C07414=1103.558,-13.554,-51.728,179.876,6.251,149.168
C07415=1103.552,-13.305,-51.741,179.876,6.255,149.169
C07416=1103.547,-13.056,-51.756,179.877,6.260,149.169
C07417=1103.543,-12.806,-51.769,179.877,6.265,149.170
C07418=1103.538,-12.557,-51.784,179.878,6.269,149.171
C07419=1103.532,-12.308,-51.798,179.878,6.273,149.172
C07420=1103.527,-12.058,-51.812,179.879,6.278,149.173
C07421=1103.522,-11.808,-51.826,179.879,6.283,149.174
C07422=1103.518,-11.558,-51.840,179.880,6.287,149.175
C07423=1103.512,-11.309,-51.854,179.880,6.292,149.175
C07424=1103.507,-11.060,-51.869,179.881,6.296,149.176
C07425=1103.502,-10.810,-51.883,179.881,6.300,149.177
C07426=1103.497,-10.560,-51.897,179.881,6.305,149.178
C07427=1103.492,-10.311,-51.911,179.882,6.310,149.179
C07428=1103.487,-10.062,-51.925,179.882,6.314,149.180
C07429=1103.482,-9.812,-51.939,179.883,6.319,149.180
C07430=1103.477,-9.562,-51.953,179.884,6.323,149.181
C07431=1103.472,-9.313,-51.968,179.884,6.327,149.182
C07432=1103.467,-9.063,-51.982,179.884,6.332,149.183
C07433=1103.463,-8.813,-51.996,179.885,6.337,149.184
C07434=1103.457,-8.564,-52.010,179.886,6.341,149.185
C07435=1103.452,-8.315,-52.024,179.886,6.346,149.186
C07436=1103.447,-8.065,-52.039,179.887,6.351,149.186
C07437=1103.442,-7.815,-52.053,179.887,6.354,149.187
C07438=1103.437,-7.565,-52.067,179.888,6.359,149.188
C07439=1103.432,-7.316,-52.081,179.888,6.364,149.189
C07440=1103.427,-7.067,-52.096,179.889,6.368,149.190
C07441=1103.422,-6.818,-52.110,179.889,6.373,149.191
C07442=1103.416,-6.568,-52.125,179.890,6.377,149.191
C07443=1103.411,-6.318,-52.140,179.891,6.382,149.192
C07444=1103.406,-6.068,-52.154,179.891,6.386,149.193
C07445=1103.401,-5.819,-52.168,179.891,6.391,149.194
C07446=1103.396,-5.570,-52.182,179.892,6.395,149.195
C07447=1103.391,-5.320,-52.197,179.893,6.400,149.196
C07448=1103.386,-5.071,-52.211,179.893,6.404,149.197
C07449=1103.382,-4.857,-52.223,179.894,6.408,149.197
C07450=1103.378,-4.642,-52.236,179.895,6.412,149.198
C07451=1103.374,-4.429,-52.248,179.895,6.416,149.199
C07452=1103.369,-4.215,-52.260,179.895,6.419,149.199
C07453=1103.365,-4.000,-52.273,179.896,6.424,149.200
C07454=1103.361,-3.787,-52.286,179.896,6.428,149.201
C07455=1103.356,-3.573,-52.298,179.897,6.431,149.201
C07456=1103.352,-3.359,-52.310,179.898,6.435,149.202
C07457=1103.347,-3.109,-52.325,179.898,6.439,149.203
C07458=1103.342,-2.860,-52.340,179.898,6.444,149.204
C07459=1103.337,-2.610,-52.354,179.899,6.448,149.205
C07460=1103.331,-2.360,-52.369,179.900,6.453,149.205
C07461=1103.327,-2.111,-52.384,179.900,6.458,149.206
C07462=1103.322,-1.861,-52.398,179.901,6.463,149.207
C07463=1103.317,-1.612,-52.412,179.902,6.467,149.208
C07464=1103.312,-1.363,-52.427,179.902,6.472,149.209
C07465=1103.307,-1.113,-52.442,179.903,6.476,149.210
C07466=1103.302,-0.863,-52.456,179.904,6.481,149.210
C07467=1103.297,-0.614,-52.471,179.904,6.485,149.211
C07468=1103.292,-0.364,-52.486,179.905,6.490,149.212
C07469=1103.287,-0.114,-52.500,179.905,6.494,149.213
C07470=1103.282,0.135,-52.516,179.906,6.498,149.214
C07471=1103.276,0.384,-52.529,179.906,6.503,149.215
C07472=1103.271,0.633,-52.544,179.907,6.508,149.216
C07473=1103.266,0.883,-52.559,179.908,6.512,149.216
C07474=1103.261,1.133,-52.574,179.908,6.517,149.217
C07475=1103.256,1.382,-52.589,179.909,6.521,149.218
C07476=1103.251,1.632,-52.603,179.910,6.526,149.219
C07477=1103.247,1.881,-52.618,179.910,6.530,149.220
C07478=1103.241,2.131,-52.633,179.911,6.535,149.220
C07479=1103.236,2.380,-52.648,179.911,6.540,149.221
C07480=1103.232,2.630,-52.662,179.912,6.544,149.222
C07481=1103.227,2.879,-52.677,179.913,6.549,149.223
C07482=1103.221,3.129,-52.692,179.913,6.554,149.224
C07483=1103.217,3.378,-52.707,179.915,6.558,149.224
C07484=1103.212,3.628,-52.721,179.915,6.563,149.225
C07485=1103.206,3.878,-52.737,179.916,6.567,149.226
C07486=1103.202,4.127,-52.751,179.916,6.572,149.227
C07487=1103.197,4.376,-52.766,179.917,6.576,149.228
C07488=1103.191,4.626,-52.782,179.918,6.581,149.229
C07489=1103.187,4.875,-52.796,179.918,6.586,149.230
C07490=1103.182,5.125,-52.811,179.919,6.590,149.230
C07491=1103.176,5.375,-52.826,179.920,6.595,149.231
C07492=1103.172,5.624,-52.841,179.920,6.600,149.232
C07493=1103.166,5.873,-52.857,179.921,6.604,149.233
C07494=1103.161,6.123,-52.871,179.922,6.609,149.234
C07495=1103.157,6.372,-52.886,179.922,6.613,149.234
C07496=1103.151,6.622,-52.901,179.923,6.618,149.235
C07497=1103.147,6.872,-52.916,179.923,6.623,149.236
C07498=1103.141,7.121,-52.932,179.924,6.627,149.237
C07499=1103.136,7.371,-52.946,179.925,6.632,149.238
C07500=1103.132,7.620,-52.961,179.926,6.636,149.239
C07501=1103.126,7.869,-52.977,179.926,6.641,149.240
C07502=1103.122,8.118,-52.992,179.927,6.645,149.240
C07503=1103.116,8.368,-53.006,179.928,6.650,149.241
C07504=1103.111,8.617,-53.021,179.929,6.656,149.242
C07505=1103.107,8.832,-53.035,179.929,6.659,149.243
C07506=1103.103,9.046,-53.047,179.929,6.663,149.244
C07507=1103.099,9.260,-53.060,179.930,6.667,149.244
C07508=1103.094,9.473,-53.074,179.930,6.671,149.245
C07509=1103.090,9.687,-53.086,179.930,6.674,149.246
C07510=1103.086,9.901,-53.100,179.930,6.678,149.247
C07511=1103.081,10.115,-53.112,179.931,6.682,149.247
C07512=1103.077,10.329,-53.126,179.931,6.686,149.248
C07513=1103.072,10.578,-53.141,179.931,6.690,149.249
C07514=1103.067,10.828,-53.156,179.932,6.694,149.250
C07515=1103.062,11.077,-53.171,179.932,6.699,149.251
C07516=1103.057,11.327,-53.186,179.932,6.703,149.252
C07517=1103.053,11.577,-53.202,179.933,6.708,149.252
C07518=1103.047,11.826,-53.217,179.933,6.712,149.253
C07519=1103.043,12.075,-53.232,179.933,6.716,149.254
C07520=1103.037,12.325,-53.248,179.934,6.721,149.255
C07521=1103.033,12.574,-53.263,179.934,6.726,149.256
C07522=1103.027,12.824,-53.278,179.934,6.730,149.257
C07523=1103.022,13.074,-53.294,179.935,6.734,149.258
C07524=1103.017,13.323,-53.309,179.936,6.739,149.259
C07525=1103.012,13.572,-53.324,179.936,6.743,149.259
C07526=1103.007,13.821,-53.339,179.936,6.747,149.260
C07527=1103.003,14.071,-53.355,179.936,6.751,149.261
C07528=1102.998,14.321,-53.370,179.937,6.756,149.262
C07529=1102.993,14.570,-53.386,179.938,6.761,149.263
C07530=1102.987,14.819,-53.401,179.937,6.765,149.264
C07531=1102.983,15.069,-53.417,179.939,6.769,149.264
C07532=1102.978,15.319,-53.432,179.939,6.774,149.265
C07533=1102.972,15.568,-53.448,179.939,6.777,149.266
C07534=1102.968,15.817,-53.463,179.940,6.782,149.267
C07535=1102.962,16.066,-53.478,179.941,6.787,149.268
C07536=1102.958,16.316,-53.494,179.941,6.790,149.269
C07537=1102.953,16.566,-53.509,179.941,6.795,149.270
C07538=1102.947,16.815,-53.525,179.942,6.800,149.270
C07539=1102.943,17.065,-53.540,179.942,6.803,149.271
C07540=1102.938,17.314,-53.556,179.943,6.808,149.272
C07541=1102.933,17.564,-53.572,179.943,6.813,149.273
C07542=1102.928,17.813,-53.587,179.944,6.816,149.273
C07543=1102.923,18.063,-53.602,179.944,6.821,149.274
C07544=1102.918,18.312,-53.618,179.944,6.825,149.275
C07545=1102.912,18.562,-53.634,179.945,6.830,149.276
C07546=1102.908,18.811,-53.649,179.946,6.834,149.277
C07547=1102.903,19.061,-53.665,179.946,6.838,149.278
C07548=1102.898,19.310,-53.680,179.947,6.842,149.278
C07549=1102.893,19.559,-53.695,179.947,6.847,149.279
C07550=1102.888,19.809,-53.711,179.947,6.851,149.280
C07551=1102.883,20.058,-53.727,179.948,6.855,149.281
C07552=1102.878,20.308,-53.743,179.949,6.860,149.282
C07553=1102.874,20.557,-53.758,179.949,6.864,149.283
C07554=1102.868,20.807,-53.774,179.950,6.868,149.283
C07555=1102.863,21.056,-53.790,179.951,6.873,149.284
C07556=1102.858,21.306,-53.805,179.951,6.876,149.285
C07557=1102.853,21.555,-53.820,179.952,6.881,149.286
C07558=1102.848,21.804,-53.837,179.952,6.884,149.286
C07559=1102.844,22.054,-53.853,179.953,6.889,149.287
C07560=1102.838,22.304,-53.868,179.954,6.893,149.288
C07561=1102.835,22.518,-53.881,179.954,6.897,149.289
C07562=1102.830,22.731,-53.895,179.954,6.900,149.289
C07563=1102.826,22.945,-53.909,179.955,6.904,149.290
C07564=1102.822,23.158,-53.922,179.955,6.908,149.291
C07565=1102.817,23.373,-53.936,179.956,6.911,149.291
C07566=1102.812,23.586,-53.949,179.956,6.915,149.292
C07567=1102.808,23.800,-53.963,179.957,6.919,149.292
C07568=1102.805,24.014,-53.977,179.958,6.922,149.293
C07569=1102.800,24.263,-53.992,179.958,6.926,149.294
C07570=1102.794,24.513,-54.008,179.959,6.931,149.295
C07571=1102.790,24.762,-54.024,179.959,6.935,149.296
C07572=1102.784,25.012,-54.040,179.960,6.939,149.296
C07573=1102.779,25.262,-54.056,179.960,6.943,149.297
C07574=1102.775,25.510,-54.072,179.961,6.948,149.298
C07575=1102.770,25.760,-54.087,179.961,6.952,149.299
C07576=1102.765,26.010,-54.103,179.962,6.956,149.299
C07577=1102.760,26.258,-54.119,179.963,6.960,149.300
C07578=1102.755,26.509,-54.135,179.963,6.964,149.301
C07579=1102.750,26.758,-54.151,179.964,6.969,149.302
C07580=1102.745,27.007,-54.167,179.965,6.972,149.302
C07581=1102.740,27.257,-54.183,179.965,6.977,149.303
C07582=1102.734,27.506,-54.199,179.966,6.981,149.304
C07583=1102.730,27.756,-54.216,179.966,6.985,149.305
C07584=1102.725,28.005,-54.231,179.967,6.989,149.305
C07585=1102.721,28.254,-54.247,179.969,6.994,149.306
C07586=1102.715,28.504,-54.263,179.968,6.997,149.307
C07587=1102.711,28.753,-54.279,179.970,7.002,149.307
C07588=1102.706,29.003,-54.295,179.971,7.006,149.308
C07589=1102.700,29.252,-54.311,179.971,7.010,149.309
C07590=1102.696,29.502,-54.327,179.972,7.014,149.310
C07591=1102.690,29.751,-54.343,179.973,7.019,149.310
C07592=1102.686,30.000,-54.360,179.973,7.022,149.311
C07593=1102.680,30.250,-54.375,179.974,7.027,149.312
C07594=1102.676,30.499,-54.392,179.974,7.030,149.313
C07595=1102.671,30.749,-54.407,179.975,7.035,149.313
C07596=1102.666,30.998,-54.424,179.976,7.039,149.314
C07597=1102.661,31.248,-54.440,179.976,7.043,149.315
C07598=1102.656,31.497,-54.456,179.977,7.047,149.315
C07599=1102.651,31.746,-54.473,179.978,7.051,149.316
C07600=1102.646,31.996,-54.489,179.979,7.055,149.317
C07601=1102.641,32.245,-54.505,179.980,7.059,149.317
C07602=1102.637,32.495,-54.521,179.980,7.064,149.318
C07603=1102.631,32.744,-54.537,179.981,7.067,149.319
C07604=1102.627,32.994,-54.553,179.982,7.072,149.320
C07605=1102.621,33.243,-54.570,179.983,7.076,149.320
C07606=1102.616,33.492,-54.587,179.983,7.080,149.321
C07607=1102.612,33.742,-54.603,179.984,7.084,149.322
C07608=1102.606,33.991,-54.619,179.985,7.089,149.322
C07609=1102.602,34.241,-54.636,179.986,7.092,149.323
C07610=1102.597,34.490,-54.651,179.987,7.096,149.324
C07611=1102.592,34.740,-54.668,179.988,7.101,149.324
C07612=1102.587,34.989,-54.683,179.988,7.104,149.325
C07613=1102.582,35.238,-54.700,179.989,7.109,149.326
C07614=1102.576,35.488,-54.717,179.990,7.113,149.326
C07615=1102.572,35.737,-54.734,179.990,7.117,149.327
C07616=1102.567,35.987,-54.750,179.991,7.121,149.328
C07617=1102.563,36.200,-54.764,179.992,7.124,149.328
C07618=1102.559,36.414,-54.778,179.993,7.128,149.329
C07619=1102.554,36.628,-54.792,179.993,7.131,149.330
C07620=1102.550,36.841,-54.806,179.994,7.134,149.330
C07621=1102.546,37.055,-54.820,179.995,7.139,149.331
C07622=1102.541,37.269,-54.834,179.996,7.142,149.331
C07623=1102.537,37.483,-54.848,179.996,7.145,149.332
C07624=1102.533,37.696,-54.862,179.997,7.149,149.332
C07625=1102.528,37.946,-54.878,179.998,7.153,149.333
C07626=1102.524,38.195,-54.895,179.998,7.157,149.334
C07627=1102.519,38.444,-54.911,180.000,7.161,149.334
C07628=1102.514,38.694,-54.928,-179.999,7.165,149.335
C07629=1102.509,38.944,-54.945,-179.999,7.169,149.336
C07630=1102.503,39.193,-54.961,-179.998,7.173,149.336
C07631=1102.499,39.442,-54.978,-179.997,7.177,149.337
C07632=1102.494,39.691,-54.994,-179.996,7.181,149.338
C07633=1102.489,39.941,-55.011,-179.995,7.185,149.338
C07634=1102.484,40.190,-55.028,-179.994,7.189,149.339
C07635=1102.479,40.439,-55.044,-179.994,7.193,149.340
C07636=1102.475,40.689,-55.061,-179.993,7.197,149.340
C07637=1102.469,40.939,-55.077,-179.992,7.202,149.341
C07638=1102.464,41.188,-55.094,-179.991,7.205,149.342
C07639=1102.460,41.437,-55.110,-179.990,7.209,149.342
C07640=1102.454,41.687,-55.128,-179.989,7.213,149.343
C07641=1102.449,41.936,-55.144,-179.988,7.217,149.343
C07642=1102.445,42.185,-55.161,-179.987,7.221,149.344
C07643=1102.440,42.435,-55.177,-179.986,7.225,149.345
C07644=1102.434,42.684,-55.194,-179.985,7.229,149.345
C07645=1102.430,42.934,-55.211,-179.984,7.233,149.346
C07646=1102.425,43.183,-55.227,-179.983,7.238,149.347
C07647=1102.420,43.433,-55.245,-179.983,7.241,149.347
C07648=1102.415,43.682,-55.261,-179.982,7.245,149.348
C07649=1102.411,43.931,-55.278,-179.980,7.249,149.348
C07650=1102.405,44.181,-55.295,-179.980,7.253,149.349
C07651=1102.400,44.430,-55.311,-179.979,7.257,149.350
C07652=1102.396,44.679,-55.328,-179.978,7.261,149.350
C07653=1102.391,44.929,-55.345,-179.977,7.266,149.351
C07654=1102.386,45.178,-55.362,-179.976,7.269,149.352
C07655=1102.380,45.428,-55.379,-179.975,7.274,149.352
C07656=1102.376,45.677,-55.395,-179.973,7.277,149.353
C07657=1102.371,45.926,-55.412,-179.973,7.281,149.353
C07658=1102.366,46.176,-55.429,-179.972,7.285,149.354
C07659=1102.361,46.424,-55.446,-179.971,7.290,149.355
C07660=1102.356,46.674,-55.464,-179.970,7.293,149.355
C07661=1102.352,46.924,-55.480,-179.969,7.297,149.356
C07662=1102.347,47.173,-55.497,-179.968,7.301,149.357
C07663=1102.341,47.422,-55.514,-179.967,7.305,149.357
C07664=1102.337,47.672,-55.531,-179.966,7.309,149.358
C07665=1102.332,47.922,-55.548,-179.965,7.313,149.359
C07666=1102.328,48.170,-55.565,-179.964,7.317,149.359
C07667=1102.322,48.420,-55.582,-179.963,7.321,149.360
C07668=1102.317,48.669,-55.599,-179.962,7.325,149.360
C07669=1102.312,48.919,-55.616,-179.961,7.329,149.361
C07670=1102.308,49.168,-55.633,-179.960,7.333,149.361
C07671=1102.303,49.417,-55.651,-179.959,7.337,149.362
C07672=1102.298,49.667,-55.667,-179.958,7.341,149.363
C07673=1102.294,49.878,-55.681,-179.957,7.344,149.363
C07674=1102.290,50.089,-55.696,-179.956,7.348,149.364
C07675=1102.285,50.301,-55.710,-179.955,7.351,149.364
C07676=1102.281,50.512,-55.726,-179.955,7.354,149.365
C07677=1102.277,50.724,-55.739,-179.953,7.358,149.365
C07678=1102.273,50.934,-55.754,-179.953,7.361,149.366
C07679=1102.269,51.146,-55.768,-179.952,7.365,149.366
C07680=1102.265,51.357,-55.783,-179.951,7.368,149.367
C07681=1102.259,51.607,-55.800,-179.950,7.372,149.367
C07682=1102.255,51.855,-55.818,-179.949,7.375,149.368
C07683=1102.250,52.105,-55.835,-179.948,7.379,149.368
C07684=1102.245,52.355,-55.852,-179.946,7.384,149.369
C07685=1102.240,52.605,-55.869,-179.945,7.388,149.370
C07686=1102.235,52.854,-55.887,-179.944,7.391,149.370
C07687=1102.231,53.103,-55.903,-179.943,7.395,149.371
C07688=1102.226,53.352,-55.921,-179.942,7.400,149.371
C07689=1101.999,43.459,-55.292,-179.978,7.245,149.347
C07690=1102.004,43.210,-55.276,-179.979,7.240,149.346
C07691=1102.009,42.960,-55.259,-179.980,7.236,149.345
C07692=1102.013,42.710,-55.242,-179.981,7.232,149.345
C07693=1102.018,42.461,-55.225,-179.981,7.228,149.344
C07694=1102.024,42.212,-55.208,-179.983,7.224,149.343
C07695=1102.028,41.962,-55.192,-179.984,7.220,149.343
C07696=1102.033,41.713,-55.175,-179.984,7.216,149.342
C07697=1102.038,41.464,-55.158,-179.985,7.212,149.341
C07698=1102.043,41.214,-55.141,-179.987,7.208,149.341
C07699=1102.047,40.965,-55.125,-179.987,7.204,149.340
C07700=1102.052,40.716,-55.108,-179.988,7.200,149.340
C07701=1102.058,40.466,-55.091,-179.989,7.196,149.339
C07702=1102.062,40.217,-55.074,-179.990,7.192,149.338
C07703=1102.068,39.967,-55.059,-179.991,7.188,149.338
C07704=1102.072,39.718,-55.042,-179.992,7.184,149.337
C07705=1102.077,39.468,-55.025,-179.992,7.180,149.336
C07706=1102.082,39.219,-55.009,-179.993,7.176,149.336
C07707=1102.087,38.970,-54.992,-179.994,7.172,149.335
C07708=1102.091,38.720,-54.975,-179.995,7.168,149.334
C07709=1102.097,38.471,-54.959,-179.996,7.164,149.334
C07710=1102.102,38.221,-54.942,-179.996,7.160,149.333
C07711=1102.107,37.972,-54.926,-179.998,7.156,149.332
C07712=1102.111,37.723,-54.909,-179.999,7.152,149.332
C07713=1102.116,37.473,-54.893,-179.999,7.148,149.331
C07714=1102.123,37.103,-54.868,180.000,7.141,149.330
C07715=1102.131,36.733,-54.844,179.999,7.136,149.329
C07716=1102.138,36.363,-54.819,179.997,7.129,149.328
C07717=1102.146,35.993,-54.795,179.996,7.123,149.327
C07718=1102.151,35.743,-54.779,179.995,7.119,149.326
C07719=1102.156,35.494,-54.762,179.995,7.116,149.326
C07720=1102.161,35.245,-54.746,179.994,7.111,149.325
C07721=1102.165,34.996,-54.729,179.993,7.107,149.324
C07722=1102.171,34.746,-54.714,179.992,7.104,149.324
C07723=1102.175,34.497,-54.697,179.991,7.099,149.323
C07724=1102.181,34.248,-54.680,179.991,7.095,149.322
C07725=1102.186,33.998,-54.664,179.990,7.091,149.322
C07726=1102.190,33.748,-54.648,179.989,7.087,149.321
C07727=1102.196,33.499,-54.632,179.988,7.082,149.320
C07728=1102.200,33.249,-54.615,179.987,7.079,149.320
C07729=1102.205,33.000,-54.599,179.986,7.075,149.319
C07730=1102.210,32.750,-54.583,179.986,7.070,149.318
C07731=1102.215,32.501,-54.567,179.985,7.066,149.317
C07732=1102.219,32.252,-54.550,179.984,7.062,149.317
C07733=1102.225,32.003,-54.534,179.983,7.058,149.316
C07734=1102.229,31.753,-54.518,179.983,7.054,149.315
C07735=1102.235,31.504,-54.502,179.982,7.050,149.314
C07736=1102.239,31.254,-54.486,179.982,7.046,149.314
C07737=1102.245,31.005,-54.470,179.981,7.042,149.313
C07738=1102.250,30.755,-54.453,179.980,7.037,149.313
C07739=1102.255,30.506,-54.437,179.980,7.034,149.312
C07740=1102.260,30.256,-54.420,179.979,7.029,149.311
C07741=1102.265,30.007,-54.405,179.978,7.025,149.310
C07742=1102.270,29.757,-54.388,179.977,7.021,149.310
C07743=1102.275,29.508,-54.373,179.977,7.017,149.309
C07744=1102.279,29.258,-54.356,179.975,7.012,149.308
C07745=1102.284,29.009,-54.341,179.975,7.009,149.307
C07746=1102.289,28.760,-54.324,179.974,7.004,149.307
C07747=1102.294,28.510,-54.309,179.973,7.000,149.306
C07748=1102.298,28.261,-54.292,179.973,6.996,149.305
C07749=1102.304,28.011,-54.276,179.972,6.992,149.304
C07750=1102.308,27.762,-54.260,179.972,6.988,149.304
C07751=1102.314,27.513,-54.244,179.971,6.984,149.303
C07752=1102.319,27.263,-54.229,179.970,6.979,149.302
C07753=1102.324,27.014,-54.212,179.970,6.976,149.302
C07754=1102.329,26.764,-54.196,179.969,6.971,149.301
C07755=1102.333,26.515,-54.180,179.968,6.967,149.300
C07756=1102.339,26.265,-54.164,179.968,6.963,149.299
C07757=1102.344,26.015,-54.148,179.967,6.958,149.298
C07758=1102.349,25.767,-54.132,179.966,6.954,149.298
C07759=1102.354,25.517,-54.116,179.966,6.951,149.297
C07760=1102.358,25.267,-54.101,179.965,6.946,149.296
C07761=1102.363,25.019,-54.085,179.965,6.942,149.296
C07762=1102.368,24.768,-54.069,179.964,6.938,149.295
C07763=1102.373,24.519,-54.053,179.963,6.933,149.294
C07764=1102.378,24.270,-54.037,179.963,6.929,149.293
C07765=1102.383,24.020,-54.021,179.962,6.925,149.292
C07766=1102.387,23.807,-54.008,179.962,6.922,149.292
C07767=1102.391,23.593,-53.994,179.961,6.918,149.291
C07768=1102.396,23.379,-53.980,179.961,6.915,149.290
C07769=1102.401,23.165,-53.967,179.960,6.911,149.290
C07770=1102.404,22.951,-53.953,179.959,6.907,149.289
C07771=1102.409,22.738,-53.939,179.959,6.903,149.289
C07772=1102.413,22.524,-53.926,179.958,6.900,149.288
C07773=1102.417,22.311,-53.913,179.958,6.896,149.287
C07774=1102.422,22.060,-53.897,179.957,6.892,149.286
C07775=1102.427,21.811,-53.881,179.957,6.888,149.286
C07776=1102.432,21.562,-53.865,179.956,6.883,149.285
C07777=1102.436,21.313,-53.850,179.956,6.880,149.284
C07778=1102.442,21.063,-53.834,179.955,6.875,149.283
C07779=1102.447,20.813,-53.818,179.955,6.870,149.282
C07780=1102.452,20.564,-53.803,179.954,6.867,149.282
C07781=1102.457,20.315,-53.786,179.954,6.862,149.281
C07782=1102.461,20.065,-53.771,179.953,6.858,149.280
C07783=1102.466,19.816,-53.755,179.953,6.854,149.279
C07784=1102.472,19.566,-53.740,179.952,6.849,149.278
C07785=1102.477,19.317,-53.724,179.952,6.846,149.278
C07786=1102.481,19.067,-53.709,179.951,6.841,149.277
C07787=1102.487,18.818,-53.693,179.951,6.836,149.276
C07788=1102.492,18.568,-53.678,179.950,6.833,149.275
C07789=1102.496,18.319,-53.662,179.950,6.828,149.274
C07790=1102.501,18.070,-53.646,179.949,6.823,149.273
C07791=1102.507,17.820,-53.630,179.949,6.820,149.273
C07792=1102.511,17.570,-53.614,179.948,6.815,149.272
C07793=1102.516,17.321,-53.599,179.948,6.810,149.271
C07794=1102.521,17.072,-53.584,179.947,6.807,149.270
C07795=1102.527,16.822,-53.568,179.947,6.802,149.270
C07796=1102.531,16.572,-53.553,179.947,6.798,149.269
C07797=1102.536,16.323,-53.537,179.946,6.794,149.268
C07798=1102.542,16.074,-53.522,179.945,6.789,149.267
C07799=1102.546,15.825,-53.507,179.945,6.785,149.266
C07800=1102.551,15.574,-53.491,179.945,6.781,149.265
C07801=1102.556,15.325,-53.475,179.944,6.776,149.264
C07802=1102.561,15.076,-53.460,179.944,6.772,149.264
C07803=1102.566,14.827,-53.445,179.943,6.768,149.263
C07804=1102.571,14.577,-53.429,179.942,6.763,149.262
C07805=1102.576,14.327,-53.414,179.943,6.759,149.261
C07806=1102.581,14.078,-53.398,179.942,6.754,149.260
C07807=1102.586,13.829,-53.383,179.941,6.750,149.259
C07808=1102.591,13.579,-53.367,179.941,6.746,149.259
C07809=1102.595,13.330,-53.352,179.940,6.742,149.258
C07810=1102.601,13.080,-53.337,179.940,6.738,149.257
C07811=1102.606,12.830,-53.322,179.940,6.733,149.256
C07812=1102.611,12.581,-53.307,179.939,6.728,149.255
C07813=1102.616,12.331,-53.291,179.939,6.724,149.254
C07814=1102.621,12.082,-53.276,179.939,6.720,149.253
C07815=1102.626,11.833,-53.260,179.938,6.715,149.252
C07816=1102.631,11.583,-53.245,179.938,6.711,149.252
C07817=1102.636,11.334,-53.230,179.938,6.706,149.251
C07818=1102.640,11.084,-53.215,179.937,6.702,149.250
C07819=1102.646,10.834,-53.199,179.937,6.698,149.249
C07820=1102.651,10.585,-53.184,179.936,6.693,149.248
C07821=1102.656,10.336,-53.169,179.936,6.689,149.247
C07822=1102.659,10.122,-53.156,179.936,6.685,149.246
C07823=1102.664,9.908,-53.142,179.935,6.681,149.246
C07824=1102.669,9.694,-53.130,179.935,6.677,149.245
C07825=1102.673,9.480,-53.117,179.935,6.674,149.244
C07826=1102.677,9.267,-53.104,179.935,6.670,149.243
C07827=1102.681,9.052,-53.090,179.935,6.666,149.243
C07828=1102.686,8.839,-53.077,179.935,6.662,149.242
C07829=1102.690,8.625,-53.065,179.934,6.658,149.241
C07830=1102.695,8.375,-53.049,179.933,6.653,149.240
C07831=1102.699,8.126,-53.034,179.933,6.649,149.239
C07832=1102.705,7.876,-53.019,179.932,6.644,149.239
C07833=1102.710,7.627,-53.005,179.931,6.640,149.238
C07834=1102.715,7.377,-52.989,179.931,6.635,149.237
C07835=1102.720,7.128,-52.974,179.930,6.630,149.236
C07836=1102.726,6.878,-52.959,179.929,6.626,149.235
C07837=1102.730,6.629,-52.944,179.928,6.621,149.234
C07838=1102.734,6.379,-52.929,179.928,6.617,149.234
C07839=1102.740,6.129,-52.914,179.927,6.612,149.233
C07840=1102.745,5.880,-52.899,179.926,6.608,149.232
C07841=1102.750,5.631,-52.883,179.926,6.603,149.231
C07842=1102.755,5.381,-52.869,179.925,6.598,149.230
C07843=1102.760,5.132,-52.854,179.924,6.594,149.230
C07844=1102.765,4.883,-52.838,179.924,6.589,149.229
C07845=1102.770,4.633,-52.824,179.923,6.584,149.228
C07846=1102.775,4.384,-52.809,179.923,6.580,149.227
C07847=1102.780,4.134,-52.794,179.922,6.575,149.226
C07848=1102.785,3.885,-52.779,179.921,6.571,149.225
C07849=1102.791,3.635,-52.764,179.921,6.566,149.224
C07850=1102.795,3.386,-52.749,179.920,6.561,149.224
C07851=1102.800,3.137,-52.734,179.919,6.557,149.223
C07852=1102.805,2.886,-52.719,179.919,6.552,149.222
C07853=1102.810,2.637,-52.704,179.918,6.547,149.221
C07854=1102.815,2.387,-52.690,179.917,6.543,149.220
C07855=1102.819,2.138,-52.675,179.916,6.538,149.220
C07856=1102.825,1.888,-52.660,179.916,6.534,149.219
C07857=1102.830,1.639,-52.645,179.915,6.529,149.218
C07858=1102.835,1.389,-52.631,179.914,6.525,149.217
C07859=1102.840,1.139,-52.616,179.914,6.520,149.216
C07860=1102.845,0.890,-52.601,179.913,6.515,149.215
C07861=1102.850,0.640,-52.587,179.912,6.511,149.215
C07862=1102.854,0.391,-52.572,179.912,6.506,149.214
C07863=1102.860,0.141,-52.557,179.911,6.502,149.213
C07864=1102.865,-0.108,-52.542,179.910,6.497,149.212
C07865=1102.870,-0.358,-52.527,179.910,6.492,149.211
C07866=1102.875,-0.607,-52.513,179.909,6.488,149.210
C07867=1102.880,-0.857,-52.498,179.909,6.483,149.209
C07868=1102.885,-1.107,-52.483,179.908,6.480,149.209
C07869=1102.890,-1.355,-52.469,179.908,6.475,149.208
C07870=1102.895,-1.605,-52.454,179.907,6.470,149.207
C07871=1102.900,-1.854,-52.440,179.906,6.466,149.206
C07872=1102.906,-2.104,-52.425,179.906,6.461,149.205
C07873=1102.911,-2.353,-52.410,179.905,6.456,149.205
C07874=1102.916,-2.603,-52.396,179.904,6.452,149.204
C07875=1102.920,-2.852,-52.381,179.904,6.447,149.203
C07876=1102.925,-3.102,-52.367,179.903,6.443,149.202
C07877=1102.930,-3.352,-52.352,179.903,6.438,149.201
C07878=1102.935,-3.565,-52.339,179.902,6.434,149.201
C07879=1102.939,-3.780,-52.327,179.902,6.431,149.200
C07880=1102.943,-3.994,-52.315,179.901,6.426,149.199
C07881=1102.948,-4.208,-52.303,179.900,6.423,149.199
C07882=1102.952,-4.421,-52.290,179.901,6.419,149.198
C07883=1102.956,-4.636,-52.278,179.900,6.415,149.197
C07884=1102.960,-4.850,-52.266,179.899,6.411,149.196
C07885=1102.964,-5.063,-52.253,179.899,6.408,149.196
C07886=1102.970,-5.313,-52.238,179.898,6.403,149.195
C07887=1102.975,-5.563,-52.224,179.898,6.398,149.194
C07888=1102.980,-5.812,-52.209,179.897,6.394,149.193
C07889=1102.985,-6.061,-52.194,179.896,6.389,149.192
C07890=1102.990,-6.310,-52.180,179.896,6.384,149.191
C07891=1102.995,-6.560,-52.166,179.895,6.380,149.190
C07892=1103.000,-6.810,-52.152,179.895,6.376,149.190
C07893=1103.005,-7.060,-52.138,179.894,6.371,149.189
C07894=1103.010,-7.309,-52.123,179.894,6.367,149.188
C07895=1103.015,-7.559,-52.109,179.893,6.362,149.187
C07896=1103.020,-7.808,-52.094,179.892,6.358,149.186
C07897=1103.025,-8.057,-52.080,179.892,6.353,149.186
C07898=1103.030,-8.307,-52.066,179.891,6.348,149.185
C07899=1103.035,-8.557,-52.052,179.891,6.344,149.184
C07900=1103.040,-8.806,-52.037,179.890,6.340,149.183
C07901=1103.045,-9.056,-52.023,179.890,6.335,149.182
C07902=1103.050,-9.306,-52.009,179.889,6.331,149.181
C07903=1103.056,-9.555,-51.995,179.889,6.326,149.180
C07904=1103.060,-9.804,-51.981,179.888,6.322,149.180
C07905=1103.065,-10.054,-51.966,179.888,6.318,149.179
C07906=1103.070,-10.304,-51.952,179.887,6.313,149.178
C07907=1103.075,-10.554,-51.938,179.887,6.308,149.177
C07908=1103.081,-10.803,-51.924,179.886,6.303,149.176
C07909=1103.086,-11.052,-51.910,179.886,6.299,149.175
C07910=1103.091,-11.302,-51.895,179.885,6.294,149.175
C07911=1103.096,-11.552,-51.881,179.885,6.291,149.174
C07912=1103.101,-11.801,-51.867,179.885,6.286,149.173
C07913=1103.106,-12.050,-51.853,179.884,6.281,149.172
C07914=1103.111,-12.300,-51.839,179.884,6.276,149.171
C07915=1103.116,-12.550,-51.824,179.883,6.272,149.170
C07916=1103.120,-12.799,-51.811,179.883,6.268,149.169
C07917=1103.126,-13.048,-51.797,179.882,6.263,149.168
C07918=1103.131,-13.298,-51.782,179.882,6.259,149.168
C07919=1103.136,-13.548,-51.768,179.881,6.254,149.167
C07920=1103.141,-13.797,-51.754,179.881,6.249,149.166
C07921=1103.146,-14.046,-51.740,179.881,6.245,149.165
C07922=1103.151,-14.296,-51.726,179.880,6.241,149.164
C07923=1103.157,-14.546,-51.712,179.879,6.236,149.163
C07924=1103.161,-14.796,-51.698,179.879,6.232,149.162
C07925=1103.166,-15.045,-51.684,179.878,6.227,149.162
C07926=1103.171,-15.295,-51.670,179.878,6.223,149.161
C07927=1103.176,-15.544,-51.656,179.878,6.218,149.160
C07928=1103.181,-15.794,-51.642,179.877,6.213,149.159
C07929=1103.187,-16.043,-51.628,179.877,6.209,149.158
C07930=1103.191,-16.293,-51.615,179.876,6.204,149.157
C07931=1103.196,-16.543,-51.600,179.877,6.200,149.156
C07932=1103.202,-16.792,-51.587,179.876,6.195,149.155
C07933=1103.207,-17.041,-51.572,179.876,6.191,149.154
C07934=1103.211,-17.255,-51.560,179.875,6.187,149.154
C07935=1103.216,-17.469,-51.548,179.875,6.182,149.153
C07936=1103.220,-17.683,-51.538,179.874,6.179,149.152
C07937=1103.224,-17.897,-51.525,179.874,6.175,149.151
C07938=1103.228,-18.112,-51.513,179.874,6.171,149.150
C07939=1103.233,-18.326,-51.501,179.873,6.167,149.150
C07940=1103.237,-18.540,-51.489,179.873,6.163,149.149
C07941=1103.241,-18.754,-51.477,179.873,6.160,149.148
C07942=1103.247,-19.003,-51.464,179.872,6.155,149.147
C07943=1103.252,-19.253,-51.450,179.872,6.150,149.146
C07944=1103.256,-19.503,-51.436,179.872,6.146,149.146
C07945=1103.262,-19.752,-51.423,179.872,6.141,149.145
C07946=1103.267,-20.002,-51.409,179.871,6.137,149.144
C07947=1103.272,-20.251,-51.395,179.871,6.132,149.143
C07948=1103.277,-20.501,-51.381,179.870,6.127,149.142
C07949=1103.282,-20.751,-51.367,179.870,6.123,149.141
C07950=1103.287,-21.000,-51.354,179.870,6.118,149.140
C07951=1103.292,-21.250,-51.340,179.870,6.114,149.139
C07952=1103.297,-21.499,-51.326,179.869,6.109,149.138
C07953=1103.302,-21.748,-51.313,179.869,6.104,149.137
C07954=1103.307,-21.998,-51.299,179.869,6.100,149.136
C07955=1103.312,-22.248,-51.285,179.868,6.095,149.135
C07956=1103.318,-22.497,-51.272,179.868,6.091,149.134
C07957=1103.322,-22.747,-51.258,179.867,6.086,149.134
C07958=1103.328,-22.996,-51.244,179.867,6.081,149.132
C07959=1103.333,-23.246,-51.231,179.868,6.077,149.132
C07960=1103.338,-23.495,-51.217,179.867,6.072,149.131
C07961=1103.343,-23.746,-51.204,179.867,6.067,149.130
C07962=1103.348,-23.995,-51.190,179.866,6.063,149.129
C07963=1103.353,-24.245,-51.177,179.866,6.058,149.128
C07964=1103.358,-24.494,-51.163,179.866,6.054,149.127
C07965=1103.364,-24.744,-51.150,179.866,6.049,149.126
C07966=1103.368,-24.993,-51.136,179.865,6.044,149.125
C07967=1103.374,-25.243,-51.123,179.865,6.039,149.124
C07968=1103.379,-25.492,-51.109,179.865,6.034,149.123
C07969=1103.384,-25.742,-51.096,179.865,6.031,149.122
C07970=1103.389,-25.991,-51.082,179.865,6.026,149.121
C07971=1103.394,-26.242,-51.068,179.865,6.021,149.120
C07972=1103.399,-26.490,-51.055,179.864,6.016,149.119
C07973=1103.404,-26.741,-51.041,179.864,6.011,149.118
C07974=1103.409,-26.989,-51.028,179.864,6.007,149.117
C07975=1103.414,-27.240,-51.015,179.863,6.003,149.116
C07976=1103.419,-27.488,-51.001,179.863,5.998,149.115
C07977=1103.424,-27.739,-50.988,179.862,5.993,149.115
C07978=1103.430,-27.988,-50.975,179.862,5.988,149.114
C07979=1103.434,-28.238,-50.961,179.862,5.984,149.113
C07980=1103.440,-28.487,-50.948,179.862,5.980,149.112
C07981=1103.444,-28.737,-50.934,179.861,5.975,149.111
C07982=1103.450,-28.986,-50.921,179.861,5.970,149.110
C07983=1103.455,-29.236,-50.908,179.861,5.966,149.109
C07984=1103.460,-29.485,-50.894,179.860,5.962,149.108
C07985=1103.465,-29.735,-50.881,179.860,5.957,149.107
C07986=1103.470,-29.985,-50.868,179.859,5.952,149.106
C07987=1103.475,-30.235,-50.854,179.860,5.948,149.105
C07988=1103.480,-30.484,-50.841,179.859,5.943,149.105
C07989=1103.485,-30.734,-50.828,179.859,5.939,149.104
C07990=1103.489,-30.948,-50.816,179.858,5.935,149.103
C07991=1103.494,-31.162,-50.805,179.858,5.931,149.102
C07992=1103.498,-31.376,-50.793,179.858,5.928,149.101
C07993=1103.503,-31.590,-50.783,179.858,5.924,149.100
C07994=1103.508,-31.804,-50.771,179.857,5.919,149.100
C07995=1103.511,-32.018,-50.760,179.857,5.916,149.099
C07996=1103.516,-32.232,-50.749,179.857,5.912,149.098
C07997=1103.521,-32.446,-50.737,179.857,5.908,149.097
C07998=1103.525,-32.696,-50.724,179.856,5.904,149.097
C07999=1103.530,-32.946,-50.711,179.856,5.900,149.096
C08000=1103.536,-33.195,-50.698,179.856,5.895,149.095
C08001=1103.540,-33.445,-50.684,179.855,5.891,149.094
C08002=1103.546,-33.694,-50.671,179.855,5.887,149.093
C08003=1103.551,-33.944,-50.658,179.855,5.882,149.092
C08004=1103.556,-34.194,-50.645,179.854,5.877,149.091
C08005=1103.561,-34.444,-50.632,179.854,5.873,149.090
C08006=1103.566,-34.693,-50.619,179.854,5.869,149.090
C08007=1103.571,-34.942,-50.606,179.853,5.864,149.089
C08008=1103.576,-35.192,-50.592,179.853,5.859,149.088
C08009=1103.581,-35.442,-50.580,179.853,5.855,149.087
C08010=1103.587,-35.692,-50.566,179.853,5.851,149.086
C08011=1103.592,-35.941,-50.554,179.852,5.846,149.085
C08012=1103.597,-36.191,-50.541,179.852,5.842,149.084
C08013=1103.602,-36.440,-50.527,179.852,5.837,149.083
C08014=1103.607,-36.690,-50.514,179.852,5.832,149.082
C08015=1103.612,-36.939,-50.502,179.852,5.828,149.081
C08016=1103.617,-37.189,-50.489,179.851,5.824,149.080
C08017=1103.622,-37.439,-50.475,179.851,5.819,149.079
C08018=1103.628,-37.688,-50.463,179.851,5.815,149.079
C08019=1103.632,-37.938,-50.450,179.850,5.810,149.078
C08020=1103.638,-38.188,-50.437,179.850,5.806,149.077
C08021=1103.643,-38.437,-50.424,179.850,5.801,149.076
C08022=1103.648,-38.687,-50.411,179.850,5.797,149.075
C08023=1103.653,-38.937,-50.398,179.849,5.792,149.074
C08024=1103.659,-39.186,-50.385,179.849,5.787,149.073
C08025=1103.663,-39.436,-50.372,179.849,5.782,149.072
C08026=1103.668,-39.685,-50.360,179.849,5.778,149.071
C08027=1103.674,-39.935,-50.346,179.849,5.774,149.070
C08028=1103.679,-40.185,-50.334,179.848,5.769,149.069
C08029=1103.684,-40.434,-50.321,179.848,5.764,149.068
C08030=1103.689,-40.684,-50.308,179.848,5.759,149.067
C08031=1103.693,-40.934,-50.295,179.848,5.755,149.066
C08032=1103.699,-41.183,-50.282,179.848,5.750,149.065
C08033=1103.704,-41.433,-50.270,179.848,5.745,149.064
C08034=1103.709,-41.682,-50.257,179.847,5.741,149.063
C08035=1103.714,-41.932,-50.244,179.847,5.735,149.062
C08036=1103.720,-42.182,-50.231,179.847,5.731,149.061
C08037=1103.725,-42.431,-50.218,179.847,5.726,149.060
C08038=1103.730,-42.681,-50.205,179.847,5.722,149.059
C08039=1103.735,-42.930,-50.193,179.847,5.716,149.058
C08040=1103.740,-43.180,-50.181,179.847,5.711,149.057
C08041=1103.745,-43.429,-50.168,179.848,5.707,149.056
C08042=1103.750,-43.680,-50.155,179.847,5.702,149.055
C08043=1103.756,-43.929,-50.142,179.848,5.698,149.054
C08044=1103.761,-44.178,-50.129,179.848,5.693,149.052
C08045=1103.766,-44.428,-50.117,179.848,5.688,149.051
C08046=1103.770,-44.642,-50.106,179.848,5.684,149.050
C08047=1103.775,-44.856,-50.095,179.848,5.680,149.049
C08048=1103.779,-45.071,-50.084,179.849,5.676,149.049
C08049=1103.783,-45.285,-50.073,179.849,5.672,149.048
C08050=1103.788,-45.499,-50.062,179.849,5.668,149.047
C08051=1103.792,-45.713,-50.052,179.849,5.664,149.046
C08052=1103.796,-45.927,-50.041,179.849,5.659,149.045
C08053=1103.801,-46.142,-50.030,179.849,5.655,149.044
C08054=1103.806,-46.392,-50.018,179.850,5.651,149.043
C08055=1103.811,-46.641,-50.005,179.850,5.646,149.042
C08056=1103.817,-46.890,-49.993,179.849,5.641,149.041
C08057=1103.821,-47.140,-49.980,179.850,5.637,149.040
C08058=1103.826,-47.390,-49.967,179.850,5.632,149.038
C08059=1103.832,-47.640,-49.955,179.850,5.628,149.038
C08060=1103.837,-47.889,-49.942,179.850,5.623,149.036
C08061=1103.842,-48.138,-49.930,179.850,5.618,149.035
C08062=1103.846,-48.388,-49.917,179.851,5.613,149.034
C08063=1103.852,-48.638,-49.905,179.850,5.609,149.033
C08064=1103.857,-48.888,-49.892,179.851,5.603,149.032
C08065=1103.862,-49.137,-49.880,179.851,5.599,149.031
C08066=1103.868,-49.387,-49.868,179.851,5.594,149.030
C08067=1103.873,-49.636,-49.855,179.851,5.589,149.029
C08068=1103.877,-49.886,-49.842,179.852,5.585,149.028
C08069=1103.883,-50.136,-49.830,179.851,5.580,149.027
C08070=1103.888,-50.385,-49.818,179.851,5.575,149.026
C08071=1103.893,-50.635,-49.805,179.852,5.571,149.024
C08072=1103.898,-50.885,-49.793,179.851,5.566,149.023
C08073=1103.903,-51.134,-49.781,179.852,5.561,149.022
C08074=1103.908,-51.384,-49.768,179.852,5.557,149.021
C08075=1103.913,-51.634,-49.756,179.852,5.552,149.020
C08076=1103.918,-51.883,-49.743,179.852,5.548,149.019
C08077=1103.924,-52.133,-49.731,179.853,5.542,149.018
C08078=1103.929,-52.383,-49.719,179.852,5.538,149.017
C08079=1103.934,-52.632,-49.706,179.853,5.533,149.016
C08080=1103.940,-52.882,-49.694,179.853,5.528,149.015
C08081=1103.945,-53.131,-49.682,179.852,5.523,149.014
C08082=1103.950,-53.382,-49.669,179.853,5.519,149.013
C08083=1103.955,-53.631,-49.657,179.853,5.514,149.011
C08084=1103.960,-53.880,-49.644,179.853,5.509,149.011
C08085=1103.965,-54.130,-49.632,179.854,5.505,149.009
C08086=1103.970,-54.380,-49.620,179.854,5.500,149.008
C08087=1103.976,-54.630,-49.608,179.853,5.495,149.007
C08088=1103.981,-54.879,-49.595,179.854,5.491,149.006
C08089=1103.986,-55.129,-49.583,179.853,5.486,149.005
C08090=1103.991,-55.378,-49.571,179.854,5.481,149.004
C08091=1103.996,-55.628,-49.560,179.854,5.477,149.003
C08092=1104.001,-55.878,-49.547,179.854,5.472,149.002
C08093=1104.006,-56.128,-49.535,179.854,5.467,149.001
C08094=1104.011,-56.377,-49.522,179.855,5.462,149.000
C08095=1104.017,-56.627,-49.510,179.854,5.458,148.999
C08096=1104.022,-56.876,-49.498,179.854,5.453,148.998
C08097=1104.027,-57.126,-49.486,179.855,5.449,148.997
C08098=1104.032,-57.375,-49.474,179.855,5.443,148.996
C08099=1104.037,-57.625,-49.462,179.855,5.438,148.994
C08100=1104.042,-57.874,-49.449,179.855,5.434,148.993
C08101=1104.048,-58.124,-49.437,179.855,5.429,148.992
C08102=1104.052,-58.339,-49.427,179.855,5.425,148.991
C08103=1104.056,-58.554,-49.417,179.855,5.421,148.990
C08104=1104.061,-58.767,-49.406,179.855,5.417,148.990
C08105=1104.065,-58.982,-49.396,179.855,5.413,148.989
C08106=1104.069,-59.196,-49.386,179.855,5.409,148.988
C08107=1104.074,-59.410,-49.375,179.855,5.405,148.987
C08108=1104.078,-59.625,-49.365,179.855,5.401,148.986
C08109=1104.082,-59.839,-49.354,179.856,5.397,148.985
C08110=1104.087,-60.089,-49.343,179.855,5.393,148.984
C08111=1104.093,-60.339,-49.331,179.855,5.387,148.983
C08112=1104.098,-60.588,-49.318,179.855,5.383,148.982
C08113=1104.103,-60.838,-49.306,179.855,5.378,148.981
C08114=1104.108,-61.088,-49.295,179.855,5.373,148.980
C08115=1104.113,-61.337,-49.282,179.854,5.368,148.979
C08116=1104.119,-61.587,-49.270,179.854,5.363,148.978
C08117=1104.124,-61.837,-49.259,179.854,5.358,148.977
C08118=1104.128,-62.086,-49.247,179.854,5.353,148.976
C08119=1104.134,-62.336,-49.235,179.854,5.348,148.975
C08120=1104.139,-62.586,-49.223,179.854,5.343,148.974
C08121=1104.144,-62.834,-49.211,179.853,5.338,148.973
C08122=1104.150,-63.084,-49.199,179.853,5.333,148.972
C08123=1104.155,-63.334,-49.187,179.853,5.329,148.971
C08124=1104.161,-63.584,-49.175,179.853,5.323,148.970
C08125=1104.165,-63.833,-49.163,179.853,5.318,148.968
C08126=1104.170,-64.083,-49.152,179.853,5.314,148.967
C08127=1104.176,-64.333,-49.140,179.853,5.308,148.966
C08128=1104.180,-64.582,-49.128,179.853,5.304,148.965
C08129=1104.186,-64.832,-49.117,179.853,5.299,148.964
C08130=1104.191,-65.081,-49.104,179.853,5.293,148.963
C08131=1104.196,-65.331,-49.093,179.852,5.289,148.962
C08132=1104.201,-65.581,-49.081,179.853,5.284,148.961
C08133=1104.207,-65.831,-49.069,179.853,5.278,148.960
C08134=1104.211,-66.081,-49.058,179.852,5.274,148.959
C08135=1104.217,-66.331,-49.046,179.852,5.268,148.958
C08136=1104.222,-66.580,-49.033,179.853,5.263,148.956
C08137=1104.227,-66.829,-49.022,179.852,5.259,148.956
C08138=1104.233,-67.079,-49.010,179.852,5.253,148.954
C08139=1104.237,-67.328,-48.999,179.852,5.248,148.953
C08140=1104.243,-67.578,-48.987,179.853,5.243,148.952
C08141=1104.248,-67.828,-48.975,179.852,5.238,148.951
C08142=1104.253,-68.078,-48.964,179.852,5.233,148.950
C08143=1104.258,-68.328,-48.952,179.852,5.228,148.949
C08144=1104.263,-68.577,-48.941,179.853,5.223,148.948
C08145=1104.268,-68.827,-48.929,179.852,5.218,148.947
C08146=1104.274,-69.076,-48.918,179.852,5.213,148.946
C08147=1104.279,-69.326,-48.906,179.852,5.208,148.944
C08148=1104.284,-69.576,-48.894,179.853,5.203,148.943
C08149=1104.289,-69.826,-48.883,179.853,5.198,148.942
C08150=1104.295,-70.076,-48.871,179.853,5.193,148.941
C08151=1104.299,-70.325,-48.859,179.853,5.188,148.940
C08152=1104.305,-70.575,-48.848,179.853,5.183,148.939
C08153=1104.310,-70.824,-48.837,179.853,5.178,148.938
C08154=1104.315,-71.074,-48.825,179.853,5.172,148.936
C08155=1104.320,-71.324,-48.814,179.853,5.167,148.935
C08156=1104.326,-71.574,-48.802,179.853,5.162,148.934
C08157=1104.330,-71.823,-48.791,179.853,5.157,148.933
C08158=1104.335,-72.037,-48.780,179.853,5.152,148.932
C08159=1104.339,-72.252,-48.770,179.853,5.148,148.931
C08160=1104.344,-72.466,-48.761,179.853,5.144,148.930
C08161=1104.349,-72.681,-48.751,179.854,5.139,148.929
C08162=1104.353,-72.895,-48.741,179.853,5.135,148.928
C08163=1104.357,-73.109,-48.731,179.853,5.131,148.927
C08164=1104.362,-73.324,-48.722,179.853,5.126,148.926
C08165=1104.366,-73.538,-48.711,179.854,5.122,148.925
C08166=1104.372,-73.787,-48.701,179.853,5.117,148.924
C08167=1104.377,-74.037,-48.689,179.854,5.112,148.923
C08168=1104.382,-74.287,-48.678,179.854,5.106,148.922
C08169=1104.387,-74.537,-48.666,179.854,5.101,148.920
C08170=1104.392,-74.786,-48.655,179.854,5.096,148.919
C08171=1104.398,-75.036,-48.643,179.854,5.091,148.918
C08172=1104.403,-75.285,-48.632,179.854,5.086,148.917
C08173=1104.408,-75.536,-48.621,179.854,5.081,148.916
C08174=1104.414,-75.785,-48.610,179.855,5.076,148.915
C08175=1104.418,-76.034,-48.598,179.855,5.071,148.913
C08176=1104.424,-76.284,-48.586,179.855,5.065,148.912
C08177=1104.428,-76.534,-48.575,179.855,5.060,148.911
C08178=1104.435,-76.784,-48.564,179.855,5.055,148.910
C08179=1104.439,-77.033,-48.553,179.855,5.050,148.909
C08180=1104.444,-77.283,-48.542,179.856,5.044,148.907
C08181=1104.450,-77.533,-48.530,179.856,5.039,148.906
C08182=1104.455,-77.783,-48.520,179.856,5.034,148.905
C08183=1104.460,-78.032,-48.508,179.856,5.029,148.904
C08184=1104.465,-78.282,-48.497,179.857,5.025,148.903
C08185=1104.471,-78.531,-48.486,179.857,5.020,148.901
C08186=1104.476,-78.781,-48.475,179.858,5.014,148.900
C08187=1104.481,-79.031,-48.463,179.858,5.009,148.899
C08188=1104.486,-79.280,-48.452,179.858,5.004,148.898
C08189=1104.492,-79.530,-48.440,179.858,4.999,148.897
C08190=1104.497,-79.780,-48.430,179.858,4.994,148.896
C08191=1104.501,-80.030,-48.418,179.858,4.989,148.894
C08192=1104.507,-80.279,-48.408,179.858,4.984,148.893
C08193=1104.512,-80.529,-48.396,179.859,4.978,148.892
C08194=1104.517,-80.779,-48.385,179.859,4.973,148.891
C08195=1104.522,-81.028,-48.374,179.859,4.968,148.889
C08196=1104.528,-81.279,-48.363,179.860,4.963,148.888
C08197=1104.533,-81.528,-48.352,179.860,4.958,148.887
C08198=1104.538,-81.778,-48.342,179.860,4.952,148.886
C08199=1104.543,-82.027,-48.330,179.861,4.948,148.885
C08200=1104.549,-82.277,-48.318,179.861,4.943,148.884
C08201=1104.554,-82.527,-48.308,179.861,4.938,148.882
C08202=1104.559,-82.776,-48.297,179.861,4.933,148.881
C08203=1104.564,-83.026,-48.287,179.861,4.927,148.880
C08204=1104.570,-83.276,-48.275,179.862,4.922,148.879
C08205=1104.575,-83.526,-48.263,179.862,4.917,148.877
C08206=1104.580,-83.775,-48.253,179.862,4.912,148.876
C08207=1104.585,-84.025,-48.242,179.863,4.907,148.875
C08208=1104.591,-84.275,-48.231,179.863,4.901,148.874
C08209=1104.596,-84.524,-48.220,179.864,4.897,148.873
C08210=1104.601,-84.774,-48.209,179.864,4.892,148.871
C08211=1104.606,-85.023,-48.198,179.864,4.887,148.870
C08212=1104.611,-85.274,-48.188,179.864,4.882,148.869
C08213=1104.616,-85.523,-48.177,179.864,4.876,148.868
C08214=1104.621,-85.737,-48.167,179.865,4.872,148.867
C08215=1104.626,-85.952,-48.158,179.865,4.868,148.866
C08216=1104.630,-86.167,-48.149,179.865,4.863,148.865
C08217=1104.635,-86.381,-48.139,179.866,4.859,148.864
C08218=1104.638,-86.595,-48.129,179.866,4.855,148.863
C08219=1104.643,-86.810,-48.121,179.866,4.850,148.862
C08220=1104.648,-87.024,-48.112,179.866,4.846,148.861
C08221=1104.652,-87.239,-48.102,179.867,4.842,148.860
C08222=1104.658,-87.488,-48.091,179.867,4.837,148.858
C08223=1104.662,-87.738,-48.080,179.868,4.831,148.857
C08224=1104.668,-87.988,-48.070,179.868,4.826,148.856
C08225=1104.673,-88.238,-48.059,179.868,4.821,148.855
C08226=1104.679,-88.487,-48.048,179.869,4.817,148.853
C08227=1104.684,-88.737,-48.037,179.869,4.812,148.852
C08228=1104.689,-88.987,-48.026,179.869,4.807,148.851
C08229=1104.694,-89.237,-48.016,179.869,4.801,148.850
C08230=1104.699,-89.486,-48.004,179.870,4.797,148.849
C08231=1104.704,-89.736,-47.994,179.870,4.792,148.848
C08232=1104.709,-89.986,-47.984,179.870,4.787,148.846
C08233=1104.715,-90.235,-47.973,179.871,4.781,148.845
C08234=1104.720,-90.485,-47.962,179.871,4.776,148.844
C08235=1104.725,-90.735,-47.952,179.872,4.772,148.843
C08236=1104.730,-90.984,-47.941,179.872,4.767,148.841
C08237=1104.736,-91.234,-47.930,179.872,4.761,148.840
C08238=1104.741,-91.484,-47.920,179.873,4.756,148.839
C08239=1104.747,-91.733,-47.908,179.873,4.752,148.838
C08240=1104.752,-91.984,-47.898,179.874,4.747,148.837
C08241=1104.757,-92.233,-47.887,179.874,4.742,148.835
C08242=1104.762,-92.483,-47.876,179.875,4.737,148.834
C08243=1104.768,-92.732,-47.866,179.875,4.732,148.833
C08244=1104.773,-92.983,-47.855,179.875,4.727,148.832
C08245=1104.778,-93.232,-47.845,179.875,4.722,148.831
C08246=1104.783,-93.482,-47.834,179.876,4.718,148.829
C08247=1104.788,-93.731,-47.824,179.876,4.712,148.828
C08248=1104.793,-93.981,-47.813,179.876,4.707,148.827
C08249=1104.799,-94.231,-47.803,179.877,4.703,148.826
C08250=1104.804,-94.481,-47.792,179.877,4.698,148.825
C08251=1104.809,-94.730,-47.781,179.878,4.693,148.823
C08252=1104.814,-94.980,-47.771,179.878,4.688,148.822
C08253=1104.820,-95.230,-47.761,179.879,4.683,148.821
C08254=1104.825,-95.480,-47.749,179.879,4.678,148.820
C08255=1104.830,-95.729,-47.739,179.880,4.674,148.819
C08256=1104.834,-95.979,-47.729,179.880,4.669,148.818
C08257=1104.840,-96.229,-47.719,179.880,4.663,148.816
C08258=1104.846,-96.478,-47.709,179.881,4.659,148.815
C08259=1104.851,-96.728,-47.698,179.881,4.654,148.814
C08260=1104.856,-96.977,-47.687,179.881,4.649,148.813
C08261=1104.861,-97.228,-47.677,179.881,4.644,148.812
C08262=1104.867,-97.477,-47.666,179.882,4.639,148.810
C08263=1104.872,-97.727,-47.656,179.882,4.634,148.809
C08264=1104.877,-97.977,-47.646,179.883,4.629,148.808
C08265=1104.883,-98.226,-47.635,179.883,4.625,148.807
C08266=1104.888,-98.477,-47.625,179.884,4.620,148.806
C08267=1104.893,-98.726,-47.614,179.884,4.614,148.804
C08268=1104.898,-98.976,-47.603,179.885,4.610,148.803
C08269=1104.904,-99.225,-47.593,179.885,4.605,148.802
C08270=1104.908,-99.440,-47.585,179.886,4.601,148.801
C08271=1104.913,-99.654,-47.577,179.886,4.597,148.800
C08272=1104.917,-99.869,-47.567,179.886,4.592,148.799
C08273=1104.922,-100.084,-47.558,179.887,4.587,148.798
C08274=1104.926,-100.298,-47.549,179.887,4.584,148.797
C08275=1104.931,-100.512,-47.540,179.887,4.580,148.796
C08276=1104.935,-100.727,-47.532,179.888,4.575,148.795
C08277=1104.939,-100.941,-47.522,179.888,4.570,148.794
C08278=1104.945,-101.191,-47.512,179.888,4.566,148.792
C08279=1104.950,-101.441,-47.502,179.889,4.561,148.791
C08280=1104.955,-101.691,-47.491,179.889,4.556,148.790
C08281=1104.961,-101.940,-47.481,179.890,4.552,148.789
C08282=1104.965,-102.190,-47.471,179.890,4.546,148.788
C08283=1104.971,-102.440,-47.461,179.890,4.541,148.786
C08284=1104.976,-102.689,-47.451,179.890,4.536,148.785
C08285=1104.981,-102.939,-47.440,179.891,4.532,148.784
C08286=1104.987,-103.189,-47.430,179.891,4.527,148.783
C08287=1104.992,-103.438,-47.420,179.892,4.521,148.782
C08288=1104.997,-103.688,-47.410,179.892,4.516,148.780
C08289=1105.002,-103.938,-47.400,179.893,4.512,148.779
C08290=1105.007,-104.188,-47.389,179.893,4.506,148.778
C08291=1105.013,-104.438,-47.380,179.894,4.501,148.777
C08292=1105.018,-104.688,-47.370,179.894,4.497,148.775
C08293=1105.023,-104.938,-47.359,179.895,4.492,148.774
C08294=1105.029,-105.187,-47.349,179.895,4.487,148.773
C08295=1105.034,-105.437,-47.339,179.895,4.481,148.772
C08296=1105.039,-105.686,-47.329,179.896,4.477,148.771
C08297=1105.044,-105.936,-47.319,179.896,4.472,148.769
C08298=1105.050,-106.186,-47.309,179.897,4.467,148.768
C08299=1105.055,-106.436,-47.298,179.897,4.462,148.767
C08300=1105.060,-106.685,-47.288,179.898,4.457,148.765
C08301=1105.065,-106.935,-47.278,179.898,4.452,148.764
C08302=1105.071,-107.185,-47.269,179.899,4.447,148.763
C08303=1105.075,-107.435,-47.259,179.899,4.442,148.762
C08304=1105.081,-107.685,-47.249,179.899,4.436,148.761
C08305=1105.087,-107.934,-47.238,179.900,4.432,148.759
C08306=1105.092,-108.184,-47.228,179.900,4.427,148.758
C08307=1105.096,-108.434,-47.218,179.900,4.422,148.757
C08308=1105.102,-108.684,-47.209,179.901,4.417,148.756
C08309=1105.108,-108.933,-47.198,179.902,4.412,148.754
C08310=1105.113,-109.183,-47.189,179.902,4.407,148.753
C08311=1105.118,-109.433,-47.178,179.902,4.402,148.752
C08312=1105.123,-109.682,-47.168,179.903,4.396,148.751
C08313=1105.129,-109.932,-47.159,179.904,4.392,148.750
C08314=1105.134,-110.182,-47.149,179.904,4.387,148.748
C08315=1105.139,-110.432,-47.138,179.904,4.382,148.747
C08316=1105.144,-110.681,-47.129,179.905,4.376,148.746
C08317=1105.150,-110.931,-47.119,179.905,4.371,148.744
C08318=1105.156,-111.181,-47.109,179.906,4.367,148.743
C08319=1105.160,-111.431,-47.099,179.906,4.362,148.742
C08320=1105.165,-111.680,-47.089,179.906,4.356,148.741
C08321=1105.171,-111.930,-47.080,179.907,4.351,148.740
C08322=1105.176,-112.180,-47.070,179.907,4.346,148.738
C08323=1105.181,-112.430,-47.059,179.908,4.341,148.737
C08324=1105.186,-112.679,-47.050,179.909,4.336,148.736
C08325=1105.192,-112.930,-47.040,179.909,4.331,148.735
C08326=1105.196,-113.144,-47.032,179.910,4.327,148.733
C08327=1105.201,-113.358,-47.023,179.909,4.322,148.732
C08328=1105.205,-113.573,-47.015,179.910,4.318,148.731
C08329=1105.210,-113.787,-47.007,179.911,4.314,148.730
C08330=1105.214,-114.003,-46.998,179.911,4.309,148.729
C08331=1105.219,-114.217,-46.989,179.911,4.305,148.728
C08332=1105.224,-114.432,-46.981,179.911,4.301,148.727
C08333=1105.228,-114.646,-46.973,179.912,4.296,148.726
C08334=1105.233,-114.895,-46.963,179.913,4.291,148.725
C08335=1105.239,-115.146,-46.953,179.913,4.286,148.723
C08336=1105.244,-115.395,-46.944,179.914,4.280,148.722
C08337=1105.250,-115.645,-46.934,179.914,4.275,148.721
C08338=1105.254,-115.895,-46.924,179.914,4.270,148.720
C08339=1105.260,-116.145,-46.914,179.915,4.266,148.718
C08340=1105.265,-116.395,-46.905,179.916,4.260,148.717
C08341=1105.270,-116.644,-46.895,179.916,4.255,148.716
C08342=1105.276,-116.894,-46.886,179.916,4.250,148.714
C08343=1105.281,-117.143,-46.876,179.917,4.244,148.713
C08344=1105.286,-117.394,-46.865,179.917,4.239,148.712
C08345=1105.291,-117.643,-46.856,179.918,4.234,148.711
C08346=1105.297,-117.893,-46.846,179.918,4.230,148.709
C08347=1105.302,-118.143,-46.837,179.919,4.224,148.708
C08348=1105.308,-118.392,-46.827,179.920,4.219,148.707
C08349=1105.313,-118.642,-46.818,179.920,4.214,148.705
C08350=1105.318,-118.892,-46.808,179.921,4.208,148.704
C08351=1105.323,-119.142,-46.799,179.921,4.203,148.703
C08352=1105.328,-119.391,-46.789,179.921,4.198,148.702
C08353=1105.334,-119.642,-46.780,179.922,4.192,148.700
C08354=1105.339,-119.891,-46.770,179.922,4.187,148.699
C08355=1105.344,-120.141,-46.761,179.923,4.183,148.698
C08356=1105.349,-120.390,-46.751,179.924,4.177,148.696
C08357=1105.355,-120.640,-46.741,179.924,4.172,148.695
C08358=1105.360,-120.890,-46.732,179.924,4.167,148.694
C08359=1105.365,-121.140,-46.723,179.925,4.162,148.692
C08360=1105.371,-121.389,-46.713,179.926,4.156,148.691
C08361=1105.376,-121.639,-46.704,179.926,4.151,148.690
C08362=1105.382,-121.889,-46.694,179.927,4.146,148.688
C08363=1105.387,-122.138,-46.685,179.927,4.141,148.687
C08364=1105.391,-122.389,-46.675,179.928,4.135,148.686
C08365=1105.397,-122.638,-46.665,179.928,4.130,148.685
C08366=1105.402,-122.888,-46.656,179.928,4.125,148.683
C08367=1105.408,-123.138,-46.647,179.929,4.119,148.682
C08368=1105.413,-123.388,-46.637,179.930,4.115,148.681
C08369=1105.418,-123.638,-46.628,179.931,4.109,148.679
C08370=1105.424,-123.887,-46.618,179.931,4.104,148.678
C08371=1105.429,-124.137,-46.609,179.932,4.099,148.676
C08372=1105.434,-124.387,-46.600,179.932,4.093,148.675
C08373=1105.440,-124.636,-46.590,179.933,4.088,148.674
C08374=1105.445,-124.886,-46.581,179.933,4.083,148.673
C08375=1105.450,-125.136,-46.572,179.934,4.077,148.671
C08376=1105.455,-125.386,-46.562,179.934,4.072,148.670
C08377=1105.461,-125.635,-46.553,179.935,4.067,148.669
C08378=1105.466,-125.885,-46.544,179.936,4.061,148.667
C08379=1105.472,-126.135,-46.535,179.936,4.056,148.666
C08380=1105.477,-126.385,-46.525,179.937,4.051,148.664
C08381=1105.482,-126.635,-46.516,179.938,4.045,148.663
C08382=1105.486,-126.849,-46.508,179.937,4.040,148.662
C08383=1105.491,-127.064,-46.500,179.938,4.036,148.661
C08384=1105.496,-127.279,-46.492,179.939,4.032,148.660
C08385=1105.500,-127.494,-46.484,179.939,4.027,148.658
C08386=1105.505,-127.708,-46.476,179.940,4.023,148.657
C08387=1105.509,-127.923,-46.468,179.940,4.017,148.656
C08388=1105.513,-128.137,-46.461,179.941,4.013,148.655
C08389=1105.518,-128.352,-46.452,179.941,4.008,148.654
C08390=1105.095,-128.343,-46.479,179.948,4.013,148.652
C08391=1105.090,-128.127,-46.486,179.948,4.017,148.654
C08392=1105.086,-127.913,-46.495,179.948,4.022,148.655
C08393=1105.082,-127.699,-46.502,179.947,4.026,148.656
C08394=1105.077,-127.484,-46.510,179.947,4.031,148.657
C08395=1105.073,-127.269,-46.518,179.946,4.036,148.658
C08396=1105.068,-127.054,-46.526,179.945,4.041,148.660
C08397=1105.064,-126.840,-46.534,179.945,4.045,148.661
C08398=1105.059,-126.625,-46.543,179.945,4.050,148.662
C08399=1105.054,-126.375,-46.552,179.944,4.055,148.663
C08400=1105.049,-126.126,-46.560,179.944,4.061,148.664
C08401=1105.043,-125.876,-46.571,179.942,4.065,148.666
C08402=1105.038,-125.626,-46.580,179.942,4.070,148.667
C08403=1105.033,-125.376,-46.588,179.941,4.076,148.669
C08404=1105.027,-125.127,-46.599,179.941,4.081,148.670
C08405=1105.022,-124.877,-46.608,179.940,4.087,148.671
C08406=1105.016,-124.627,-46.617,179.940,4.092,148.673
C08407=1105.011,-124.378,-46.627,179.939,4.097,148.674
C08408=1105.006,-124.128,-46.636,179.939,4.102,148.675
C08409=1105.000,-123.878,-46.645,179.938,4.108,148.676
C08410=1104.995,-123.628,-46.655,179.937,4.113,148.678
C08411=1104.990,-123.378,-46.664,179.937,4.118,148.679
C08412=1104.985,-123.129,-46.674,179.936,4.124,148.681
C08413=1104.979,-122.879,-46.683,179.936,4.129,148.682
C08414=1104.974,-122.630,-46.693,179.935,4.135,148.683
C08415=1104.969,-122.380,-46.702,179.935,4.140,148.685
C08416=1104.964,-122.129,-46.711,179.935,4.145,148.686
C08417=1104.958,-121.880,-46.721,179.934,4.150,148.687
C08418=1104.953,-121.630,-46.730,179.934,4.156,148.688
C08419=1104.948,-121.380,-46.740,179.932,4.160,148.690
C08420=1104.943,-121.130,-46.749,179.932,4.165,148.691
C08421=1104.937,-120.881,-46.759,179.932,4.171,148.692
C08422=1104.932,-120.631,-46.768,179.931,4.176,148.694
C08423=1104.927,-120.382,-46.778,179.931,4.181,148.695
C08424=1104.921,-120.132,-46.787,179.930,4.186,148.696
C08425=1104.916,-119.882,-46.797,179.929,4.192,148.698
C08426=1104.911,-119.631,-46.807,179.929,4.197,148.699
C08427=1104.906,-119.382,-46.817,179.928,4.203,148.700
C08428=1104.900,-119.132,-46.826,179.928,4.207,148.702
C08429=1104.895,-118.883,-46.836,179.927,4.212,148.703
C08430=1104.889,-118.633,-46.845,179.927,4.217,148.704
C08431=1104.884,-118.383,-46.855,179.926,4.223,148.705
C08432=1104.879,-118.133,-46.864,179.926,4.228,148.707
C08433=1104.874,-117.883,-46.874,179.926,4.233,148.708
C08434=1104.869,-117.634,-46.884,179.925,4.239,148.709
C08435=1104.864,-117.384,-46.893,179.925,4.244,148.711
C08436=1104.858,-117.134,-46.904,179.924,4.248,148.712
C08437=1104.853,-116.885,-46.912,179.923,4.254,148.713
C08438=1104.847,-116.635,-46.923,179.923,4.259,148.714
C08439=1104.842,-116.386,-46.932,179.922,4.264,148.716
C08440=1104.837,-116.135,-46.942,179.922,4.269,148.717
C08441=1104.831,-115.885,-46.952,179.921,4.275,148.718
C08442=1104.826,-115.635,-46.961,179.921,4.280,148.720
C08443=1104.821,-115.386,-46.971,179.920,4.284,148.721
C08444=1104.816,-115.137,-46.981,179.920,4.289,148.722
C08445=1104.810,-114.887,-46.991,179.919,4.295,148.723
C08446=1104.806,-114.637,-47.000,179.919,4.300,148.725
C08447=1104.801,-114.422,-47.009,179.919,4.304,148.726
C08448=1104.796,-114.207,-47.018,179.918,4.308,148.727
C08449=1104.791,-113.993,-47.026,179.918,4.313,148.728
C08450=1104.787,-113.778,-47.034,179.917,4.317,148.729
C08451=1104.782,-113.564,-47.043,179.917,4.321,148.730
C08452=1104.778,-113.350,-47.051,179.917,4.327,148.731
C08453=1104.773,-113.135,-47.059,179.916,4.331,148.732
C08454=1104.769,-112.921,-47.068,179.915,4.335,148.733
C08455=1104.764,-112.670,-47.078,179.915,4.340,148.735
C08456=1104.758,-112.420,-47.088,179.915,4.345,148.736
C08457=1104.753,-112.171,-47.097,179.915,4.350,148.737
C08458=1104.747,-111.921,-47.108,179.913,4.355,148.738
C08459=1104.743,-111.671,-47.118,179.913,4.360,148.740
C08460=1104.737,-111.421,-47.127,179.913,4.365,148.741
C08461=1104.732,-111.172,-47.137,179.912,4.371,148.742
C08462=1104.727,-110.923,-47.147,179.912,4.376,148.743
C08463=1104.722,-110.672,-47.157,179.911,4.380,148.744
C08464=1104.716,-110.423,-47.168,179.911,4.386,148.746
C08465=1104.711,-110.173,-47.177,179.910,4.391,148.747
C08466=1104.705,-109.923,-47.187,179.910,4.396,148.748
C08467=1104.700,-109.673,-47.197,179.909,4.400,148.750
C08468=1104.696,-109.424,-47.207,179.909,4.405,148.751
C08469=1104.690,-109.174,-47.217,179.909,4.410,148.752
C08470=1104.684,-108.924,-47.227,179.909,4.416,148.753
C08471=1104.680,-108.674,-47.237,179.908,4.421,148.755
C08472=1104.674,-108.425,-47.247,179.907,4.426,148.756
C08473=1104.669,-108.175,-47.257,179.907,4.431,148.757
C08474=1104.664,-107.925,-47.268,179.906,4.436,148.758
C08475=1104.659,-107.676,-47.277,179.906,4.441,148.759
C08476=1104.653,-107.426,-47.287,179.905,4.445,148.761
C08477=1104.648,-107.177,-47.298,179.905,4.450,148.762
C08478=1104.642,-106.926,-47.308,179.905,4.456,148.763
C08479=1104.637,-106.676,-47.317,179.904,4.461,148.765
C08480=1104.632,-106.427,-47.327,179.903,4.465,148.766
C08481=1104.627,-106.177,-47.338,179.903,4.471,148.767
C08482=1104.621,-105.927,-47.348,179.903,4.476,148.768
C08483=1104.616,-105.678,-47.358,179.903,4.481,148.769
C08484=1104.611,-105.428,-47.368,179.902,4.485,148.771
C08485=1104.606,-105.178,-47.379,179.902,4.490,148.772
C08486=1104.600,-104.929,-47.389,179.901,4.496,148.773
C08487=1104.596,-104.679,-47.399,179.901,4.501,148.774
C08488=1104.590,-104.429,-47.409,179.900,4.505,148.775
C08489=1104.585,-104.180,-47.419,179.900,4.510,148.777
C08490=1104.580,-103.929,-47.430,179.900,4.515,148.778
C08491=1104.574,-103.680,-47.440,179.899,4.520,148.779
C08492=1104.569,-103.431,-47.450,179.898,4.525,148.780
C08493=1104.564,-103.180,-47.460,179.898,4.530,148.782
C08494=1104.559,-102.931,-47.470,179.898,4.536,148.783
C08495=1104.554,-102.681,-47.481,179.897,4.540,148.784
C08496=1104.548,-102.431,-47.491,179.897,4.545,148.785
C08497=1104.543,-102.182,-47.501,179.897,4.550,148.786
C08498=1104.538,-101.931,-47.511,179.896,4.555,148.788
C08499=1104.533,-101.682,-47.522,179.896,4.560,148.789
C08500=1104.527,-101.432,-47.532,179.895,4.565,148.790
C08501=1104.522,-101.182,-47.542,179.895,4.570,148.791
C08502=1104.516,-100.933,-47.553,179.894,4.574,148.792
C08503=1104.512,-100.718,-47.561,179.895,4.579,148.793
C08504=1104.508,-100.504,-47.570,179.894,4.583,148.795
C08505=1104.503,-100.289,-47.579,179.893,4.587,148.795
C08506=1104.499,-100.075,-47.588,179.893,4.591,148.796
C08507=1104.494,-99.861,-47.597,179.892,4.596,148.798
C08508=1104.490,-99.645,-47.606,179.893,4.600,148.799
C08509=1104.486,-99.431,-47.615,179.892,4.604,148.800
C08510=1104.481,-99.217,-47.623,179.892,4.609,148.801
C08511=1104.475,-98.967,-47.633,179.891,4.614,148.802
C08512=1104.470,-98.717,-47.644,179.891,4.618,148.803
C08513=1104.465,-98.467,-47.654,179.890,4.623,148.804
C08514=1104.460,-98.218,-47.665,179.890,4.628,148.806
C08515=1104.455,-97.968,-47.676,179.889,4.633,148.807
C08516=1104.450,-97.718,-47.686,179.889,4.638,148.808
C08517=1104.444,-97.468,-47.696,179.889,4.643,148.809
C08518=1104.438,-97.219,-47.707,179.888,4.647,148.810
C08519=1104.433,-96.969,-47.717,179.888,4.653,148.812
C08520=1104.428,-96.720,-47.728,179.888,4.658,148.813
C08521=1104.423,-96.469,-47.739,179.887,4.663,148.814
C08522=1104.417,-96.220,-47.749,179.887,4.667,148.815
C08523=1104.412,-95.970,-47.760,179.886,4.672,148.816
C08524=1104.407,-95.720,-47.770,179.886,4.677,148.817
C08525=1104.402,-95.471,-47.781,179.885,4.682,148.819
C08526=1104.397,-95.221,-47.791,179.885,4.687,148.820
C08527=1104.392,-94.971,-47.802,179.885,4.692,148.821
C08528=1104.386,-94.721,-47.812,179.884,4.696,148.822
C08529=1104.381,-94.472,-47.823,179.884,4.702,148.823
C08530=1104.376,-94.222,-47.834,179.884,4.707,148.825
C08531=1104.370,-93.972,-47.844,179.883,4.711,148.826
C08532=1104.365,-93.722,-47.854,179.883,4.716,148.827
C08533=1104.360,-93.473,-47.865,179.883,4.721,148.828
C08534=1104.355,-93.223,-47.876,179.882,4.726,148.829
C08535=1104.349,-92.974,-47.886,179.882,4.731,148.831
C08536=1104.345,-92.724,-47.897,179.881,4.736,148.832
C08537=1104.339,-92.474,-47.908,179.881,4.741,148.833
C08538=1104.334,-92.224,-47.918,179.880,4.745,148.834
C08539=1104.329,-91.974,-47.929,179.880,4.751,148.835
C08540=1104.324,-91.725,-47.940,179.880,4.756,148.837
C08541=1104.319,-91.475,-47.950,179.879,4.760,148.838
C08542=1104.313,-91.226,-47.961,179.879,4.765,148.839
C08543=1104.308,-90.976,-47.972,179.879,4.770,148.840
C08544=1104.303,-90.726,-47.982,179.879,4.776,148.841
C08545=1104.298,-90.476,-47.993,179.877,4.780,148.843
C08546=1104.292,-90.227,-48.003,179.877,4.785,148.844
C08547=1104.287,-89.977,-48.015,179.877,4.791,148.845
C08548=1104.281,-89.727,-48.025,179.877,4.796,148.846
C08549=1104.276,-89.477,-48.036,179.877,4.801,148.848
C08550=1104.271,-89.228,-48.047,179.876,4.805,148.849
C08551=1104.266,-88.978,-48.058,179.876,4.810,148.850
C08552=1104.261,-88.728,-48.069,179.876,4.815,148.851
C08553=1104.256,-88.479,-48.079,179.875,4.821,148.852
C08554=1104.251,-88.228,-48.090,179.875,4.826,148.853
C08555=1104.246,-87.980,-48.101,179.874,4.830,148.855
C08556=1104.240,-87.729,-48.112,179.874,4.835,148.856
C08557=1104.235,-87.480,-48.123,179.873,4.841,148.857
C08558=1104.230,-87.230,-48.133,179.873,4.846,148.858
C08559=1104.225,-87.016,-48.142,179.873,4.850,148.859
C08560=1104.221,-86.801,-48.152,179.873,4.854,148.860
C08561=1104.216,-86.587,-48.162,179.873,4.859,148.862
C08562=1104.212,-86.373,-48.170,179.872,4.863,148.862
C08563=1104.207,-86.158,-48.180,179.872,4.867,148.864
C08564=1104.203,-85.944,-48.189,179.872,4.872,148.865
C08565=1104.199,-85.729,-48.199,179.872,4.876,148.866
C08566=1104.194,-85.514,-48.208,179.871,4.880,148.867
C08567=1104.189,-85.265,-48.219,179.871,4.885,148.868
C08568=1104.183,-85.016,-48.230,179.871,4.891,148.869
C08569=1104.178,-84.765,-48.241,179.870,4.896,148.870
C08570=1104.173,-84.516,-48.252,179.870,4.901,148.871
C08571=1104.168,-84.266,-48.262,179.870,4.906,148.873
C08572=1104.163,-84.016,-48.274,179.869,4.910,148.874
C08573=1104.157,-83.767,-48.285,179.869,4.915,148.875
C08574=1104.152,-83.517,-48.296,179.868,4.921,148.876
C08575=1104.148,-83.267,-48.307,179.868,4.926,148.878
C08576=1104.141,-83.018,-48.318,179.868,4.931,148.879
C08577=1104.137,-82.768,-48.329,179.868,4.936,148.880
C08578=1104.132,-82.518,-48.340,179.868,4.942,148.881
C08579=1104.126,-82.269,-48.351,179.868,4.947,148.882
C08580=1104.121,-82.019,-48.363,179.867,4.952,148.883
C08581=1104.116,-81.769,-48.373,179.867,4.957,148.885
C08582=1104.111,-81.520,-48.384,179.866,4.961,148.886
C08583=1104.105,-81.270,-48.396,179.866,4.966,148.887
C08584=1104.100,-81.020,-48.407,179.866,4.972,148.888
C08585=1104.095,-80.771,-48.418,179.865,4.977,148.890
C08586=1104.090,-80.521,-48.429,179.865,4.982,148.891
C08587=1104.085,-80.270,-48.440,179.865,4.987,148.892
C08588=1104.079,-80.022,-48.451,179.865,4.992,148.893
C08589=1104.075,-79.772,-48.462,179.865,4.998,148.894
C08590=1104.069,-79.521,-48.473,179.865,5.003,148.896
C08591=1104.064,-79.272,-48.484,179.864,5.008,148.897
C08592=1104.058,-79.022,-48.496,179.864,5.013,148.898
C08593=1104.053,-78.773,-48.507,179.864,5.018,148.899
C08594=1104.048,-78.523,-48.518,179.864,5.023,148.900
C08595=1104.042,-78.273,-48.530,179.864,5.028,148.901
C08596=1104.038,-78.024,-48.541,179.864,5.034,148.903
C08597=1104.033,-77.774,-48.552,179.864,5.039,148.904
C08598=1104.027,-77.524,-48.563,179.862,5.043,148.905
C08599=1104.022,-77.275,-48.574,179.862,5.049,148.906
C08600=1104.017,-77.025,-48.586,179.862,5.054,148.908
C08601=1104.012,-76.775,-48.597,179.862,5.059,148.909
C08602=1104.007,-76.526,-48.608,179.862,5.064,148.910
C08603=1104.001,-76.276,-48.619,179.862,5.069,148.911
C08604=1103.996,-76.026,-48.631,179.861,5.074,148.912
C08605=1103.991,-75.776,-48.643,179.861,5.079,148.913
C08606=1103.985,-75.527,-48.654,179.861,5.085,148.915
C08607=1103.980,-75.277,-48.665,179.861,5.090,148.916
C08608=1103.975,-75.028,-48.677,179.861,5.095,148.917
C08609=1103.971,-74.778,-48.688,179.861,5.100,148.918
C08610=1103.965,-74.527,-48.699,179.860,5.105,148.919
C08611=1103.960,-74.278,-48.710,179.860,5.110,148.920
C08612=1103.954,-74.029,-48.722,179.860,5.115,148.922
C08613=1103.949,-73.779,-48.733,179.860,5.120,148.923
C08614=1103.944,-73.529,-48.745,179.860,5.126,148.924
C08615=1103.939,-73.315,-48.755,179.860,5.130,148.925
C08616=1103.936,-73.100,-48.764,179.860,5.134,148.926
C08617=1103.931,-72.887,-48.775,179.860,5.138,148.927
C08618=1103.927,-72.672,-48.785,179.860,5.143,148.928
C08619=1103.922,-72.458,-48.794,179.859,5.147,148.929
C08620=1103.917,-72.243,-48.804,179.860,5.152,148.930
C08621=1103.912,-72.029,-48.814,179.860,5.156,148.931
C08622=1103.909,-71.815,-48.824,179.859,5.161,148.932
C08623=1103.903,-71.565,-48.835,179.859,5.165,148.933
C08624=1103.898,-71.315,-48.846,179.859,5.170,148.934
C08625=1103.893,-71.065,-48.858,179.859,5.175,148.935
C08626=1103.887,-70.815,-48.870,179.859,5.181,148.936
C08627=1103.883,-70.566,-48.882,179.859,5.186,148.938
C08628=1103.877,-70.316,-48.894,179.859,5.191,148.939
C08629=1103.873,-70.067,-48.905,179.858,5.196,148.940
C08630=1103.867,-69.818,-48.917,179.858,5.201,148.941
C08631=1103.862,-69.568,-48.928,179.859,5.206,148.942
C08632=1103.856,-69.318,-48.940,179.859,5.211,148.943
C08633=1103.852,-69.068,-48.951,179.858,5.216,148.944
C08634=1103.846,-68.818,-48.963,179.858,5.221,148.945
C08635=1103.841,-68.569,-48.975,179.858,5.226,148.947
C08636=1103.836,-68.319,-48.986,179.858,5.231,148.948
C08637=1103.831,-68.069,-48.998,179.858,5.236,148.949
C08638=1103.826,-67.820,-49.009,179.858,5.241,148.950
C08639=1103.820,-67.570,-49.021,179.858,5.247,148.951
C08640=1103.815,-67.320,-49.033,179.858,5.251,148.952
C08641=1103.810,-67.071,-49.045,179.858,5.256,148.953
C08642=1103.805,-66.821,-49.057,179.858,5.262,148.954
C08643=1103.799,-66.571,-49.068,179.858,5.267,148.956
C08644=1103.795,-66.322,-49.080,179.859,5.271,148.956
C08645=1103.789,-66.072,-49.092,179.858,5.277,148.958
C08646=1103.784,-65.822,-49.104,179.858,5.282,148.959
C08647=1103.779,-65.573,-49.116,179.859,5.286,148.960
C08648=1103.774,-65.323,-49.127,179.859,5.292,148.961
C08649=1103.769,-65.073,-49.139,179.858,5.297,148.962
C08650=1103.763,-64.824,-49.150,179.859,5.301,148.963
C08651=1103.758,-64.574,-49.162,179.859,5.307,148.964
C08652=1103.753,-64.325,-49.175,179.859,5.312,148.965
C08653=1103.748,-64.075,-49.186,179.859,5.316,148.966
C08654=1103.743,-63.825,-49.198,179.859,5.322,148.967
C08655=1103.737,-63.575,-49.210,179.859,5.326,148.968
C08656=1103.733,-63.326,-49.222,179.859,5.331,148.969
C08657=1103.727,-63.076,-49.234,179.859,5.337,148.971
C08658=1103.722,-62.826,-49.246,179.859,5.341,148.972
C08659=1103.717,-62.577,-49.258,179.859,5.346,148.973
C08660=1103.712,-62.327,-49.269,179.860,5.351,148.974
C08661=1103.707,-62.077,-49.281,179.860,5.356,148.975
C08662=1103.701,-61.828,-49.293,179.860,5.361,148.976
C08663=1103.696,-61.578,-49.306,179.860,5.366,148.977
C08664=1103.691,-61.329,-49.317,179.860,5.371,148.978
C08665=1103.686,-61.079,-49.329,179.861,5.376,148.979
C08666=1103.681,-60.829,-49.342,179.860,5.381,148.980
C08667=1103.676,-60.579,-49.353,179.861,5.386,148.981
C08668=1103.670,-60.330,-49.366,179.861,5.391,148.982
C08669=1103.666,-60.080,-49.377,179.861,5.395,148.983
C08670=1103.660,-59.831,-49.389,179.862,5.400,148.984
C08671=1103.656,-59.616,-49.400,179.861,5.404,148.985
C08672=1103.652,-59.402,-49.411,179.861,5.408,148.986
C08673=1103.647,-59.188,-49.420,179.862,5.413,148.987
C08674=1103.643,-58.974,-49.431,179.861,5.417,148.988
C08675=1103.639,-58.759,-49.441,179.861,5.421,148.989
C08676=1103.634,-58.545,-49.452,179.861,5.425,148.989
C08677=1103.629,-58.331,-49.463,179.861,5.429,148.990
C08678=1103.625,-58.116,-49.473,179.861,5.433,148.991
C08679=1103.620,-57.867,-49.485,179.861,5.437,148.992
C08680=1103.615,-57.617,-49.497,179.861,5.442,148.993
C08681=1103.610,-57.368,-49.509,179.860,5.447,148.995
C08682=1103.605,-57.118,-49.521,179.861,5.452,148.995
C08683=1103.600,-56.868,-49.534,179.860,5.457,148.997
C08684=1103.594,-56.618,-49.546,179.860,5.461,148.998
C08685=1103.589,-56.369,-49.558,179.860,5.466,148.999
C08686=1103.584,-56.119,-49.570,179.860,5.471,149.000
C08687=1103.579,-55.870,-49.583,179.860,5.475,149.001
C08688=1103.574,-55.620,-49.594,179.860,5.480,149.002
C08689=1103.569,-55.370,-49.607,179.860,5.485,149.003
C08690=1103.564,-55.120,-49.619,179.860,5.489,149.004
C08691=1103.559,-54.871,-49.631,179.859,5.494,149.005
C08692=1103.553,-54.621,-49.643,179.860,5.499,149.006
C08693=1103.548,-54.372,-49.656,179.859,5.503,149.007
C08694=1103.543,-54.122,-49.669,179.859,5.508,149.008
C08695=1103.538,-53.872,-49.680,179.859,5.513,149.009
C08696=1103.533,-53.623,-49.693,179.859,5.517,149.011
C08697=1103.527,-53.373,-49.705,179.859,5.522,149.012
C08698=1103.523,-53.123,-49.718,179.859,5.527,149.013
C08699=1103.517,-52.874,-49.730,179.858,5.532,149.014
C08700=1103.512,-52.624,-49.742,179.859,5.536,149.015
C08701=1103.507,-52.375,-49.755,179.859,5.541,149.016
C08702=1103.502,-52.125,-49.767,179.858,5.546,149.017
C08703=1103.496,-51.875,-49.779,179.858,5.550,149.018
C08704=1103.491,-51.626,-49.792,179.858,5.556,149.019
C08705=1103.486,-51.375,-49.804,179.858,5.560,149.020
C08706=1103.481,-51.126,-49.817,179.858,5.565,149.021
C08707=1103.476,-50.877,-49.829,179.858,5.570,149.022
C08708=1103.471,-50.627,-49.841,179.857,5.574,149.023
C08709=1103.466,-50.377,-49.854,179.858,5.579,149.024
C08710=1103.461,-50.128,-49.867,179.858,5.584,149.026
C08711=1103.456,-49.878,-49.879,179.857,5.588,149.027
C08712=1103.451,-49.628,-49.891,179.857,5.593,149.028
C08713=1103.445,-49.379,-49.904,179.857,5.598,149.029
C08714=1103.440,-49.130,-49.917,179.857,5.602,149.030
C08715=1103.435,-48.880,-49.929,179.857,5.608,149.031
C08716=1103.430,-48.630,-49.941,179.857,5.612,149.032
C08717=1103.425,-48.380,-49.954,179.856,5.617,149.033
C08718=1103.420,-48.131,-49.967,179.856,5.622,149.034
C08719=1103.415,-47.881,-49.979,179.856,5.626,149.035
C08720=1103.410,-47.632,-49.991,179.856,5.631,149.036
C08721=1103.404,-47.382,-50.004,179.856,5.636,149.038
C08722=1103.400,-47.132,-50.017,179.855,5.640,149.039
C08723=1103.394,-46.882,-50.029,179.856,5.645,149.040
C08724=1103.389,-46.633,-50.042,179.856,5.650,149.041
C08725=1103.383,-46.384,-50.054,179.855,5.654,149.042
C08726=1103.379,-46.133,-50.067,179.855,5.659,149.043
C08727=1103.374,-45.920,-50.078,179.855,5.663,149.044
C08728=1103.370,-45.706,-50.088,179.855,5.667,149.045
C08729=1103.366,-45.491,-50.100,179.854,5.671,149.046
C08730=1103.362,-45.277,-50.110,179.854,5.675,149.047
C08731=1103.357,-45.063,-50.121,179.855,5.680,149.048
C08732=1103.352,-44.849,-50.132,179.855,5.684,149.049
C08733=1103.348,-44.635,-50.143,179.854,5.688,149.049
C08734=1103.344,-44.420,-50.154,179.854,5.692,149.050
C08735=1103.338,-44.171,-50.167,179.854,5.696,149.052
C08736=1103.333,-43.921,-50.179,179.854,5.701,149.052
C08737=1103.329,-43.671,-50.192,179.854,5.706,149.054
C08738=1103.323,-43.422,-50.205,179.853,5.710,149.055
C08739=1103.318,-43.172,-50.217,179.853,5.715,149.056
C08740=1103.313,-42.922,-50.230,179.854,5.720,149.057
C08741=1103.308,-42.673,-50.243,179.853,5.725,149.058
C08742=1103.302,-42.423,-50.256,179.853,5.730,149.059
C08743=1103.297,-42.174,-50.268,179.853,5.734,149.060
C08744=1103.293,-41.924,-50.281,179.853,5.739,149.061
C08745=1103.288,-41.675,-50.294,179.854,5.744,149.062
C08746=1103.282,-41.425,-50.307,179.853,5.749,149.063
C08747=1103.277,-41.175,-50.320,179.854,5.753,149.064
C08748=1103.272,-40.926,-50.333,179.854,5.758,149.065
C08749=1103.267,-40.676,-50.345,179.854,5.763,149.066
C08750=1103.261,-40.427,-50.358,179.854,5.767,149.067
C08751=1103.257,-40.177,-50.371,179.854,5.772,149.068
C08752=1103.252,-39.927,-50.384,179.854,5.777,149.069
C08753=1103.246,-39.678,-50.397,179.855,5.782,149.070
C08754=1103.241,-39.428,-50.410,179.854,5.786,149.071
C08755=1103.236,-39.178,-50.423,179.855,5.790,149.072
C08756=1103.231,-38.929,-50.435,179.855,5.795,149.073
C08757=1103.226,-38.679,-50.449,179.855,5.800,149.074
C08758=1103.221,-38.429,-50.461,179.855,5.804,149.075
C08759=1103.215,-38.180,-50.474,179.856,5.809,149.076
C08760=1103.211,-37.930,-50.487,179.856,5.814,149.077
C08761=1103.205,-37.680,-50.500,179.856,5.818,149.078
C08762=1103.201,-37.431,-50.514,179.856,5.822,149.079
C08763=1103.196,-37.182,-50.526,179.857,5.827,149.079
C08764=1103.190,-36.932,-50.540,179.857,5.832,149.080
C08765=1103.185,-36.682,-50.553,179.857,5.836,149.081
C08766=1103.180,-36.433,-50.565,179.858,5.840,149.082
C08767=1103.174,-36.183,-50.578,179.858,5.845,149.083
C08768=1103.170,-35.933,-50.591,179.858,5.849,149.084
C08769=1103.165,-35.684,-50.604,179.858,5.854,149.085
C08770=1103.160,-35.434,-50.618,179.859,5.859,149.086
C08771=1103.155,-35.185,-50.631,179.859,5.862,149.087
C08772=1103.149,-34.935,-50.644,179.859,5.867,149.088
C08773=1103.144,-34.685,-50.657,179.859,5.872,149.089
C08774=1103.139,-34.436,-50.670,179.859,5.876,149.089
C08775=1103.134,-34.186,-50.684,179.860,5.881,149.090
C08776=1103.129,-33.937,-50.697,179.860,5.885,149.091
C08777=1103.123,-33.687,-50.710,179.860,5.889,149.092
C08778=1103.119,-33.437,-50.723,179.861,5.894,149.093
C08779=1103.114,-33.188,-50.735,179.861,5.898,149.094
C08780=1103.109,-32.938,-50.750,179.861,5.902,149.095
C08781=1103.103,-32.689,-50.762,179.862,5.907,149.096
C08782=1103.098,-32.438,-50.776,179.862,5.912,149.097
C08783=1103.094,-32.225,-50.787,179.862,5.916,149.097
C08784=1103.089,-32.011,-50.798,179.862,5.919,149.098
C08785=1103.085,-31.797,-50.809,179.863,5.923,149.099
C08786=1103.081,-31.583,-50.821,179.863,5.927,149.100
C08787=1103.077,-31.369,-50.832,179.864,5.931,149.100
C08788=1103.072,-31.155,-50.844,179.864,5.935,149.101
C08789=1103.067,-30.940,-50.855,179.864,5.938,149.102
C08790=1103.064,-30.726,-50.866,179.864,5.942,149.103
C08791=1103.058,-30.476,-50.880,179.865,5.947,149.104
C08792=1103.053,-30.227,-50.893,179.865,5.951,149.105
C08793=1103.048,-29.977,-50.907,179.865,5.955,149.105
C08794=1103.043,-29.728,-50.919,179.865,5.960,149.106
C08795=1103.038,-29.478,-50.934,179.866,5.965,149.107
C08796=1103.033,-29.229,-50.946,179.866,5.970,149.108
C08797=1103.028,-28.978,-50.960,179.866,5.974,149.109
C08798=1103.023,-28.730,-50.973,179.867,5.978,149.110
C08799=1103.018,-28.479,-50.987,179.867,5.983,149.111
C08800=1103.013,-28.230,-50.999,179.868,5.988,149.112
C08801=1103.008,-27.980,-51.014,179.867,5.992,149.113
C08802=1103.003,-27.731,-51.026,179.868,5.996,149.114
C08803=1102.998,-27.481,-51.040,179.868,6.001,149.114
C08804=1102.992,-27.232,-51.053,179.869,6.006,149.115
C08805=1102.987,-26.982,-51.067,179.869,6.011,149.116
C08806=1102.982,-26.733,-51.081,179.869,6.014,149.117
C08807=1102.977,-26.483,-51.094,179.870,6.019,149.118
C08808=1102.972,-26.234,-51.107,179.870,6.024,149.119
C08809=1102.967,-25.984,-51.121,179.871,6.029,149.120
C08810=1102.962,-25.734,-51.135,179.871,6.034,149.121
C08811=1102.957,-25.485,-51.148,179.871,6.039,149.122
C08812=1102.952,-25.235,-51.162,179.871,6.042,149.123
C08813=1102.946,-24.986,-51.175,179.871,6.047,149.124
C08814=1102.942,-24.736,-51.188,179.871,6.052,149.125
C08815=1102.936,-24.487,-51.202,179.872,6.057,149.126
C08816=1102.931,-24.237,-51.216,179.872,6.062,149.127
C08817=1102.926,-23.988,-51.229,179.872,6.066,149.128
C08818=1102.921,-23.737,-51.243,179.872,6.071,149.129
C08819=1102.916,-23.488,-51.257,179.873,6.075,149.130
C08820=1102.911,-23.239,-51.270,179.873,6.080,149.131
C08821=1102.906,-22.989,-51.284,179.874,6.085,149.131
C08822=1102.900,-22.740,-51.298,179.873,6.089,149.132
C08823=1102.896,-22.490,-51.311,179.873,6.094,149.134
C08824=1102.891,-22.240,-51.325,179.874,6.099,149.134
C08825=1102.885,-21.991,-51.339,179.874,6.103,149.135
C08826=1102.881,-21.741,-51.352,179.874,6.107,149.136
C08827=1102.875,-21.492,-51.366,179.875,6.112,149.137
C08828=1102.870,-21.242,-51.379,179.875,6.117,149.138
C08829=1102.866,-20.992,-51.393,179.876,6.122,149.139
C08830=1102.860,-20.743,-51.407,179.876,6.126,149.140
C08831=1102.855,-20.493,-51.421,179.876,6.131,149.141
C08832=1102.850,-20.243,-51.435,179.876,6.135,149.142
C08833=1102.845,-19.995,-51.448,179.877,6.140,149.143
C08834=1102.840,-19.745,-51.462,179.877,6.145,149.144
C08835=1102.835,-19.494,-51.476,179.878,6.149,149.145
C08836=1102.829,-19.245,-51.490,179.877,6.153,149.146
C08837=1102.825,-18.996,-51.504,179.878,6.158,149.146
C08838=1102.820,-18.746,-51.517,179.878,6.163,149.147
C08839=1102.816,-18.532,-51.529,179.879,6.166,149.148
C08840=1102.811,-18.318,-51.541,179.879,6.170,149.149
C08841=1102.807,-18.104,-51.553,179.880,6.175,149.150
C08842=1102.802,-17.890,-51.565,179.880,6.179,149.150
C08843=1102.798,-17.676,-51.577,179.880,6.182,149.151
C08844=1102.794,-17.462,-51.589,179.880,6.186,149.152
C08845=1102.789,-17.249,-51.601,179.881,6.190,149.153
C08846=1102.785,-17.035,-51.613,179.881,6.194,149.153
C08847=1102.780,-16.784,-51.626,179.882,6.199,149.154
C08848=1102.775,-16.535,-51.641,179.882,6.203,149.155
C08849=1102.770,-16.286,-51.654,179.882,6.207,149.156
C08850=1102.765,-16.036,-51.668,179.883,6.212,149.157
C08851=1102.760,-15.786,-51.683,179.883,6.217,149.158
C08852=1102.755,-15.537,-51.696,179.883,6.221,149.159
C08853=1102.749,-15.287,-51.710,179.883,6.225,149.160
C08854=1102.744,-15.037,-51.724,179.884,6.230,149.161
C08855=1102.739,-14.788,-51.739,179.884,6.235,149.162
C08856=1102.735,-14.539,-51.752,179.885,6.239,149.162
C08857=1102.730,-14.289,-51.766,179.885,6.244,149.163
C08858=1102.725,-14.040,-51.780,179.886,6.248,149.164
C08859=1102.720,-13.790,-51.795,179.886,6.252,149.165
C08860=1102.714,-13.541,-51.809,179.887,6.257,149.166
C08861=1102.709,-13.291,-51.823,179.887,6.262,149.167
C08862=1102.704,-13.041,-51.837,179.888,6.267,149.168
C08863=1102.699,-12.792,-51.851,179.888,6.271,149.168
C08864=1102.694,-12.542,-51.866,179.888,6.275,149.169
C08865=1102.689,-12.293,-51.880,179.889,6.280,149.170
C08866=1102.685,-12.044,-51.893,179.890,6.284,149.171
C08867=1102.680,-11.794,-51.908,179.890,6.289,149.172
C08868=1102.675,-11.544,-51.922,179.890,6.293,149.173
C08869=1102.669,-11.295,-51.936,179.891,6.298,149.174
C08870=1102.664,-11.045,-51.950,179.891,6.302,149.175
C08871=1102.659,-10.796,-51.964,179.892,6.307,149.175
C08872=1102.654,-10.546,-51.979,179.893,6.311,149.176
C08873=1102.649,-10.296,-51.993,179.893,6.316,149.177
C08874=1102.644,-10.047,-52.007,179.893,6.320,149.178
C08875=1102.639,-9.798,-52.021,179.893,6.325,149.179
C08876=1102.634,-9.548,-52.035,179.894,6.329,149.179
C08877=1102.629,-9.298,-52.050,179.895,6.334,149.180
C08878=1102.624,-9.048,-52.064,179.895,6.339,149.181
C08879=1102.619,-8.799,-52.078,179.896,6.343,149.182
C08880=1102.614,-8.549,-52.092,179.896,6.347,149.183
C08881=1102.608,-8.300,-52.106,179.897,6.352,149.184
C08882=1102.603,-8.050,-52.121,179.897,6.356,149.185
C08883=1102.599,-7.801,-52.136,179.898,6.361,149.186
C08884=1102.594,-7.552,-52.150,179.898,6.366,149.186
C08885=1102.589,-7.302,-52.164,179.899,6.370,149.187
C08886=1102.584,-7.052,-52.178,179.900,6.375,149.188
C08887=1102.579,-6.802,-52.193,179.900,6.379,149.189
C08888=1102.573,-6.553,-52.207,179.900,6.383,149.190
C08889=1102.568,-6.304,-52.222,179.901,6.388,149.190
C08890=1102.563,-6.054,-52.237,179.902,6.392,149.191
C08891=1102.558,-5.805,-52.251,179.902,6.397,149.192
C08892=1102.553,-5.555,-52.265,179.903,6.402,149.193
C08893=1102.548,-5.305,-52.279,179.904,6.406,149.194
C08894=1102.544,-5.056,-52.294,179.904,6.410,149.195
C08895=1102.539,-4.842,-52.306,179.905,6.414,149.195
C08896=1102.535,-4.628,-52.318,179.905,6.418,149.196
C08897=1102.530,-4.415,-52.332,179.905,6.422,149.197
C08898=1102.526,-4.200,-52.344,179.906,6.426,149.198
C08899=1102.521,-3.986,-52.356,179.906,6.430,149.198
C08900=1102.517,-3.773,-52.369,179.907,6.433,149.199
C08901=1102.513,-3.559,-52.381,179.908,6.438,149.200
C08902=1102.509,-3.345,-52.394,179.908,6.442,149.201
C08903=1102.504,-3.095,-52.408,179.909,6.446,149.201
C08904=1102.499,-2.845,-52.423,179.909,6.451,149.202
C08905=1102.494,-2.595,-52.438,179.910,6.455,149.203
C08906=1102.488,-2.347,-52.452,179.911,6.460,149.204
C08907=1102.483,-2.097,-52.466,179.911,6.464,149.205
C08908=1102.479,-1.848,-52.481,179.912,6.469,149.205
C08909=1102.473,-1.598,-52.496,179.912,6.473,149.206
C08910=1102.468,-1.348,-52.511,179.913,6.477,149.207
C08911=1102.463,-1.099,-52.526,179.913,6.482,149.208
C08912=1102.459,-0.850,-52.540,179.914,6.487,149.209
C08913=1102.454,-0.600,-52.554,179.915,6.491,149.209
C08914=1102.448,-0.351,-52.570,179.915,6.496,149.210
C08915=1102.443,-0.101,-52.584,179.916,6.500,149.211
C08916=1102.439,0.148,-52.599,179.917,6.505,149.212
C08917=1102.434,0.398,-52.613,179.917,6.509,149.213
C08918=1102.428,0.647,-52.629,179.918,6.514,149.214
C08919=1102.423,0.897,-52.643,179.918,6.519,149.215
C08920=1102.419,1.146,-52.658,179.919,6.523,149.215
C08921=1102.413,1.396,-52.673,179.920,6.528,149.216
C08922=1102.408,1.645,-52.688,179.920,6.533,149.217
C08923=1102.403,1.895,-52.702,179.921,6.537,149.218
C08924=1102.399,2.144,-52.717,179.922,6.542,149.219
C08925=1102.393,2.394,-52.732,179.923,6.546,149.220
C08926=1102.388,2.643,-52.747,179.924,6.551,149.220
C08927=1102.383,2.893,-52.761,179.924,6.555,149.221
C08928=1102.378,3.142,-52.777,179.925,6.560,149.222
C08929=1102.374,3.393,-52.792,179.925,6.565,149.223
C08930=1102.369,3.642,-52.807,179.926,6.569,149.224
C08931=1102.363,3.892,-52.821,179.927,6.574,149.224
C08932=1102.359,4.141,-52.836,179.927,6.579,149.225
C08933=1102.353,4.390,-52.852,179.928,6.583,149.226
C08934=1102.348,4.640,-52.866,179.929,6.588,149.227
C08935=1102.344,4.889,-52.881,179.929,6.592,149.228
C08936=1102.338,5.139,-52.896,179.930,6.597,149.229
C08937=1102.333,5.388,-52.911,179.931,6.601,149.229
C08938=1102.329,5.637,-52.926,179.931,6.606,149.230
C08939=1102.323,5.887,-52.941,179.932,6.611,149.231
C08940=1102.318,6.136,-52.956,179.932,6.615,149.232
C08941=1102.314,6.387,-52.972,179.933,6.620,149.233
C08942=1102.309,6.636,-52.986,179.934,6.624,149.234
C08943=1102.303,6.886,-53.002,179.935,6.629,149.234
C08944=1102.299,7.135,-53.017,179.936,6.634,149.235
C08945=1102.294,7.384,-53.032,179.936,6.638,149.236
C08946=1102.288,7.634,-53.047,179.937,6.643,149.237
C08947=1102.284,7.883,-53.062,179.937,6.648,149.238
C08948=1102.278,8.132,-53.077,179.938,6.652,149.238
C08949=1102.274,8.382,-53.093,179.939,6.657,149.239
C08950=1102.268,8.632,-53.108,179.939,6.661,149.240
C08951=1102.264,8.846,-53.120,179.940,6.665,149.241
C08952=1102.260,9.060,-53.134,179.940,6.670,149.242
C08953=1102.256,9.273,-53.147,179.941,6.673,149.242
C08954=1102.251,9.487,-53.160,179.941,6.677,149.243
C08955=1102.247,9.701,-53.172,179.941,6.681,149.244
C08956=1102.243,9.915,-53.185,179.941,6.684,149.245
C08957=1102.239,10.129,-53.199,179.941,6.688,149.246
C08958=1102.234,10.342,-53.212,179.941,6.692,149.246
C08959=1102.229,10.592,-53.227,179.942,6.697,149.247
C08960=1102.224,10.841,-53.242,179.942,6.701,149.248
C08961=1102.220,11.091,-53.258,179.942,6.705,149.249
C08962=1102.215,11.341,-53.272,179.943,6.710,149.250
C08963=1102.209,11.590,-53.288,179.943,6.713,149.251
C08964=1102.204,11.839,-53.304,179.944,6.718,149.252
C08965=1102.199,12.089,-53.319,179.944,6.723,149.252
C08966=1102.195,12.339,-53.335,179.944,6.727,149.253
C08967=1102.190,12.588,-53.350,179.945,6.731,149.254
C08968=1102.184,12.837,-53.365,179.945,6.736,149.255
C08969=1102.180,13.086,-53.380,179.945,6.740,149.256
C08970=1102.174,13.336,-53.396,179.946,6.745,149.257
C08971=1102.170,13.586,-53.412,179.947,6.749,149.258
C08972=1102.165,13.835,-53.427,179.946,6.753,149.259
C08973=1102.159,14.085,-53.442,179.948,6.758,149.259
C08974=1102.154,14.334,-53.457,179.947,6.762,149.260
C08975=1102.150,14.584,-53.473,179.948,6.766,149.261
C08976=1102.144,14.833,-53.488,179.949,6.771,149.262
C08977=1102.140,15.083,-53.503,179.949,6.775,149.263
C08978=1102.134,15.332,-53.519,179.949,6.780,149.264
C08979=1102.130,15.582,-53.535,179.950,6.784,149.264
C08980=1102.125,15.831,-53.550,179.950,6.788,149.265
C08981=1102.120,16.081,-53.565,179.951,6.793,149.266
C08982=1102.114,16.330,-53.581,179.951,6.796,149.267
C08983=1102.110,16.579,-53.597,179.952,6.801,149.268
C08984=1102.105,16.828,-53.612,179.952,6.805,149.269
C08985=1102.100,17.078,-53.628,179.952,6.809,149.270
C08986=1102.096,17.328,-53.643,179.953,6.814,149.270
C08987=1102.090,17.577,-53.659,179.954,6.818,149.271
C08988=1102.085,17.826,-53.675,179.954,6.822,149.272
C08989=1102.080,18.076,-53.690,179.954,6.827,149.273
C08990=1102.075,18.326,-53.706,179.955,6.831,149.273
C08991=1102.070,18.575,-53.721,179.955,6.835,149.274
C08992=1102.065,18.824,-53.737,179.956,6.840,149.275
C08993=1102.060,19.075,-53.753,179.956,6.843,149.276
C08994=1102.056,19.323,-53.768,179.957,6.848,149.277
C08995=1102.050,19.572,-53.784,179.957,6.853,149.278
C08996=1102.045,19.823,-53.800,179.958,6.856,149.278
C08997=1102.040,20.072,-53.816,179.958,6.861,149.279
C08998=1102.035,20.321,-53.831,179.958,6.865,149.280
C08999=1102.031,20.571,-53.846,179.959,6.869,149.281
C09000=1102.025,20.820,-53.863,179.960,6.874,149.282
C09001=1102.020,21.069,-53.878,179.960,6.877,149.282
C09002=1102.016,21.319,-53.894,179.961,6.882,149.283
C09003=1102.011,21.569,-53.909,179.962,6.887,149.284
C09004=1102.005,21.818,-53.925,179.962,6.890,149.285
C09005=1102.001,22.067,-53.942,179.963,6.895,149.286
C09006=1101.995,22.317,-53.957,179.964,6.899,149.286
C09007=1101.989,22.645,-53.977,179.964,6.904,149.287
C09008=1101.983,22.972,-53.999,179.964,6.910,149.289
C09009=1101.977,23.300,-54.019,179.966,6.916,149.289
C09010=1101.970,23.628,-54.040,179.966,6.922,149.290
C09011=1101.965,23.876,-54.056,179.967,6.925,149.291
C09012=1101.959,24.126,-54.072,179.967,6.930,149.292
C09013=1101.955,24.376,-54.088,179.968,6.933,149.293
C09014=1101.950,24.624,-54.104,179.968,6.938,149.294
C09015=1101.946,24.874,-54.120,179.969,6.942,149.294
C09016=1101.940,25.124,-54.135,179.969,6.946,149.295
C09017=1101.935,25.373,-54.151,179.970,6.951,149.296
C09018=1101.930,25.623,-54.167,179.971,6.955,149.296
C09019=1101.925,25.872,-54.183,179.971,6.959,149.297
C09020=1101.920,26.122,-54.200,179.972,6.963,149.298
C09021=1101.915,26.371,-54.215,179.972,6.967,149.299
C09022=1101.910,26.621,-54.231,179.973,6.971,149.300
C09023=1101.905,26.870,-54.247,179.975,6.976,149.300
C09024=1101.900,27.119,-54.263,179.974,6.980,149.301
C09025=1101.895,27.369,-54.280,179.976,6.984,149.302
C09026=1101.891,27.618,-54.295,179.976,6.989,149.303
C09027=1101.886,27.867,-54.311,179.977,6.992,149.303
C09028=1101.881,28.117,-54.327,179.978,6.996,149.304
C09029=1101.876,28.366,-54.344,179.978,7.000,149.305
C09030=1101.871,28.616,-54.359,179.979,7.005,149.305
C09031=1101.866,28.866,-54.375,179.980,7.009,149.306
C09032=1101.861,29.114,-54.392,179.980,7.013,149.307
C09033=1101.856,29.365,-54.407,179.981,7.017,149.308
C09034=1101.851,29.613,-54.424,179.982,7.021,149.308
C09035=1101.846,29.863,-54.440,179.982,7.025,149.309
C09036=1101.841,30.112,-54.456,179.983,7.030,149.310
C09037=1101.837,30.362,-54.473,179.984,7.034,149.311
C09038=1101.831,30.611,-54.488,179.984,7.038,149.311
C09039=1101.827,30.861,-54.505,179.985,7.042,149.312
C09040=1101.822,31.110,-54.521,179.985,7.046,149.313
C09041=1101.817,31.360,-54.537,179.986,7.050,149.313
C09042=1101.812,31.609,-54.553,179.987,7.054,149.314
C09043=1101.806,31.859,-54.570,179.987,7.058,149.315
C09044=1101.801,32.108,-54.586,179.988,7.063,149.316
C09045=1101.797,32.358,-54.602,179.990,7.067,149.316
C09046=1101.792,32.606,-54.619,179.990,7.070,149.317
C09047=1101.787,32.857,-54.635,179.991,7.075,149.318
C09048=1101.782,33.105,-54.651,179.992,7.079,149.318
C09049=1101.777,33.355,-54.668,179.992,7.083,149.319
C09050=1101.772,33.604,-54.683,179.993,7.087,149.320
C09051=1101.545,23.775,-54.093,179.972,6.926,149.290
C09052=1101.553,23.412,-54.071,179.971,6.921,149.289
C09053=1101.560,23.050,-54.048,179.969,6.914,149.288
C09054=1101.567,22.687,-54.024,179.969,6.908,149.287
C09055=1101.574,22.324,-54.002,179.968,6.902,149.286
C09056=1101.579,22.074,-53.986,179.967,6.898,149.285
C09057=1101.584,21.825,-53.970,179.967,6.894,149.284
C09058=1101.590,21.575,-53.954,179.966,6.889,149.283
C09059=1101.594,21.325,-53.938,179.966,6.885,149.282
C09060=1101.599,21.076,-53.923,179.965,6.881,149.282
C09061=1101.604,20.828,-53.907,179.965,6.876,149.281
C09062=1101.609,20.577,-53.891,179.964,6.873,149.280
C09063=1101.614,20.328,-53.875,179.964,6.868,149.279
C09064=1101.620,20.079,-53.860,179.963,6.863,149.278
C09065=1101.624,19.829,-53.844,179.963,6.860,149.278
C09066=1101.629,19.580,-53.828,179.962,6.855,149.277
C09067=1101.634,19.331,-53.812,179.962,6.851,149.276
C09068=1101.639,19.081,-53.796,179.961,6.847,149.275
C09069=1101.644,18.831,-53.781,179.961,6.842,149.274
C09070=1101.649,18.582,-53.766,179.961,6.838,149.273
C09071=1101.654,18.332,-53.750,179.960,6.834,149.273
C09072=1101.659,18.083,-53.734,179.959,6.829,149.272
C09073=1101.663,17.834,-53.718,179.959,6.826,149.271
C09074=1101.668,17.584,-53.703,179.958,6.821,149.270
C09075=1101.674,17.335,-53.687,179.958,6.817,149.269
C09076=1101.679,17.085,-53.671,179.958,6.813,149.269
C09077=1101.683,16.835,-53.656,179.957,6.808,149.268
C09078=1101.688,16.586,-53.640,179.957,6.804,149.267
C09079=1101.694,16.337,-53.625,179.956,6.800,149.266
C09080=1101.699,16.087,-53.610,179.956,6.795,149.265
C09081=1101.703,15.837,-53.594,179.956,6.791,149.264
C09082=1101.709,15.588,-53.578,179.955,6.787,149.264
C09083=1101.713,15.339,-53.563,179.955,6.783,149.263
C09084=1101.718,15.089,-53.547,179.954,6.778,149.262
C09085=1101.724,14.839,-53.532,179.954,6.773,149.261
C09086=1101.728,14.590,-53.517,179.954,6.770,149.260
C09087=1101.734,14.341,-53.501,179.953,6.765,149.259
C09088=1101.738,14.091,-53.485,179.952,6.761,149.259
C09089=1101.743,13.842,-53.470,179.952,6.757,149.258
C09090=1101.748,13.592,-53.455,179.951,6.752,149.257
C09091=1101.753,13.343,-53.440,179.952,6.748,149.256
C09092=1101.758,13.093,-53.424,179.951,6.743,149.255
C09093=1101.763,12.844,-53.408,179.950,6.739,149.254
C09094=1101.768,12.595,-53.393,179.950,6.735,149.253
C09095=1101.773,12.345,-53.378,179.950,6.730,149.252
C09096=1101.778,12.096,-53.363,179.949,6.726,149.252
C09097=1101.783,11.846,-53.347,179.949,6.722,149.251
C09098=1101.788,11.597,-53.331,179.948,6.717,149.250
C09099=1101.793,11.347,-53.316,179.948,6.713,149.249
C09100=1101.798,11.097,-53.301,179.948,6.708,149.248
C09101=1101.803,10.848,-53.286,179.947,6.704,149.247
C09102=1101.808,10.598,-53.270,179.947,6.700,149.246
C09103=1101.812,10.349,-53.255,179.947,6.695,149.246
C09104=1101.817,10.136,-53.242,179.947,6.691,149.245
C09105=1101.821,9.922,-53.229,179.947,6.688,149.244
C09106=1101.826,9.708,-53.215,179.947,6.684,149.243
C09107=1101.830,9.495,-53.203,179.946,6.680,149.242
C09108=1101.835,9.280,-53.190,179.946,6.676,149.242
C09109=1101.839,9.066,-53.177,179.945,6.672,149.241
C09110=1101.842,8.852,-53.164,179.945,6.668,149.240
C09111=1101.847,8.639,-53.150,179.945,6.665,149.239
C09112=1101.852,8.390,-53.135,179.944,6.660,149.238
C09113=1101.857,8.140,-53.120,179.943,6.656,149.238
C09114=1101.862,7.890,-53.105,179.943,6.651,149.237
C09115=1101.867,7.640,-53.090,179.942,6.646,149.236
C09116=1101.872,7.391,-53.075,179.942,6.641,149.235
C09117=1101.877,7.142,-53.059,179.941,6.637,149.234
C09118=1101.882,6.892,-53.045,179.940,6.632,149.234
C09119=1101.887,6.643,-53.029,179.940,6.628,149.233
C09120=1101.892,6.394,-53.014,179.939,6.623,149.232
C09121=1101.898,6.144,-52.999,179.938,6.619,149.231
C09122=1101.902,5.894,-52.984,179.937,6.613,149.230
C09123=1101.906,5.645,-52.969,179.936,6.608,149.229
C09124=1101.912,5.395,-52.954,179.936,6.604,149.228
C09125=1101.917,5.146,-52.939,179.935,6.599,149.228
C09126=1101.922,4.896,-52.924,179.934,6.595,149.227
C09127=1101.927,4.647,-52.909,179.934,6.590,149.226
C09128=1101.932,4.398,-52.894,179.933,6.586,149.225
C09129=1101.937,4.148,-52.879,179.932,6.581,149.224
C09130=1101.942,3.898,-52.864,179.932,6.576,149.224
C09131=1101.947,3.649,-52.849,179.931,6.572,149.223
C09132=1101.952,3.399,-52.834,179.930,6.567,149.222
C09133=1101.956,3.149,-52.819,179.930,6.563,149.221
C09134=1101.962,2.900,-52.804,179.929,6.558,149.220
C09135=1101.967,2.650,-52.789,179.928,6.554,149.220
C09136=1101.971,2.401,-52.774,179.927,6.549,149.219
C09137=1101.977,2.151,-52.759,179.927,6.544,149.218
C09138=1101.982,1.902,-52.744,179.926,6.539,149.217
C09139=1101.987,1.652,-52.730,179.925,6.535,149.216
C09140=1101.992,1.403,-52.715,179.925,6.530,149.215
C09141=1101.997,1.153,-52.700,179.924,6.526,149.214
C09142=1102.002,0.904,-52.685,179.924,6.522,149.214
C09143=1102.007,0.655,-52.671,179.923,6.517,149.213
C09144=1102.012,0.405,-52.655,179.923,6.513,149.212
C09145=1102.017,0.155,-52.641,179.922,6.508,149.211
C09146=1102.022,-0.094,-52.626,179.921,6.504,149.210
C09147=1102.027,-0.343,-52.612,179.921,6.499,149.209
C09148=1102.032,-0.593,-52.596,179.920,6.494,149.209
C09149=1102.037,-0.842,-52.582,179.919,6.490,149.208
C09150=1102.042,-1.092,-52.568,179.919,6.485,149.207
C09151=1102.047,-1.341,-52.553,179.918,6.480,149.206
C09152=1102.052,-1.591,-52.538,179.917,6.476,149.205
C09153=1102.057,-1.840,-52.523,179.917,6.471,149.205
C09154=1102.062,-2.090,-52.509,179.916,6.467,149.204
C09155=1102.067,-2.340,-52.494,179.916,6.462,149.203
C09156=1102.072,-2.589,-52.479,179.915,6.459,149.202
C09157=1102.077,-2.839,-52.464,179.915,6.454,149.201
C09158=1102.082,-3.089,-52.450,179.914,6.449,149.200
C09159=1102.087,-3.338,-52.435,179.913,6.445,149.200
C09160=1102.091,-3.552,-52.423,179.913,6.440,149.199
C09161=1102.095,-3.765,-52.410,179.912,6.437,149.198
C09162=1102.101,-3.979,-52.398,179.912,6.433,149.197
C09163=1102.104,-4.194,-52.385,179.911,6.429,149.197
C09164=1102.109,-4.407,-52.373,179.911,6.425,149.196
C09165=1102.113,-4.621,-52.361,179.910,6.422,149.195
C09166=1102.117,-4.834,-52.348,179.910,6.417,149.194
C09167=1102.121,-5.049,-52.336,179.909,6.413,149.194
C09168=1102.127,-5.298,-52.322,179.909,6.409,149.193
C09169=1102.132,-5.548,-52.307,179.908,6.404,149.192
C09170=1102.137,-5.797,-52.292,179.908,6.400,149.191
C09171=1102.142,-6.047,-52.277,179.907,6.396,149.190
C09172=1102.147,-6.297,-52.263,179.907,6.391,149.190
C09173=1102.152,-6.546,-52.249,179.906,6.387,149.189
C09174=1102.157,-6.796,-52.235,179.905,6.382,149.188
C09175=1102.161,-7.045,-52.220,179.905,6.377,149.187
C09176=1102.166,-7.295,-52.205,179.904,6.372,149.186
C09177=1102.172,-7.544,-52.191,179.904,6.369,149.186
C09178=1102.177,-7.793,-52.177,179.903,6.364,149.185
C09179=1102.182,-8.043,-52.163,179.903,6.359,149.184
C09180=1102.187,-8.292,-52.148,179.902,6.355,149.183
C09181=1102.191,-8.542,-52.134,179.901,6.350,149.182
C09182=1102.197,-8.792,-52.119,179.901,6.346,149.181
C09183=1102.202,-9.042,-52.104,179.901,6.342,149.180
C09184=1102.208,-9.291,-52.091,179.900,6.337,149.179
C09185=1102.213,-9.540,-52.076,179.900,6.332,149.179
C09186=1102.218,-9.790,-52.062,179.899,6.328,149.178
C09187=1102.223,-10.040,-52.048,179.898,6.323,149.177
C09188=1102.227,-10.290,-52.033,179.898,6.319,149.176
C09189=1102.232,-10.539,-52.019,179.898,6.315,149.175
C09190=1102.238,-10.788,-52.005,179.898,6.310,149.174
C09191=1102.243,-11.037,-51.990,179.897,6.306,149.174
C09192=1102.247,-11.287,-51.977,179.896,6.301,149.173
C09193=1102.252,-11.536,-51.962,179.896,6.296,149.172
C09194=1102.257,-11.786,-51.948,179.895,6.291,149.171
C09195=1102.262,-12.035,-51.934,179.895,6.288,149.170
C09196=1102.267,-12.285,-51.920,179.895,6.283,149.169
C09197=1102.272,-12.535,-51.906,179.894,6.279,149.168
C09198=1102.277,-12.784,-51.891,179.893,6.274,149.168
C09199=1102.282,-13.034,-51.877,179.893,6.269,149.167
C09200=1102.288,-13.283,-51.863,179.893,6.265,149.166
C09201=1102.293,-13.533,-51.849,179.892,6.260,149.165
C09202=1102.298,-13.783,-51.835,179.892,6.256,149.164
C09203=1102.303,-14.033,-51.821,179.891,6.251,149.163
C09204=1102.308,-14.282,-51.807,179.890,6.247,149.162
C09205=1102.313,-14.531,-51.793,179.890,6.243,149.161
C09206=1102.318,-14.781,-51.779,179.890,6.238,149.161
C09207=1102.323,-15.031,-51.765,179.889,6.233,149.160
C09208=1102.328,-15.280,-51.751,179.889,6.229,149.159
C09209=1102.333,-15.529,-51.737,179.888,6.224,149.158
C09210=1102.338,-15.779,-51.722,179.889,6.220,149.157
C09211=1102.343,-16.029,-51.708,179.888,6.215,149.156
C09212=1102.349,-16.278,-51.695,179.888,6.210,149.155
C09213=1102.353,-16.528,-51.681,179.887,6.206,149.154
C09214=1102.358,-16.778,-51.667,179.887,6.202,149.153
C09215=1102.363,-17.027,-51.653,179.887,6.197,149.152
C09216=1102.367,-17.241,-51.641,179.886,6.194,149.152
C09217=1102.372,-17.455,-51.629,179.886,6.189,149.151
C09218=1102.376,-17.669,-51.617,179.885,6.185,149.150
C09219=1102.381,-17.883,-51.605,179.885,6.182,149.150
C09220=1102.385,-18.097,-51.593,179.885,6.178,149.149
C09221=1102.389,-18.310,-51.581,179.884,6.174,149.148
C09222=1102.394,-18.525,-51.570,179.884,6.170,149.147
C09223=1102.398,-18.739,-51.558,179.884,6.166,149.146
C09224=1102.403,-18.989,-51.543,179.883,6.161,149.145
C09225=1102.407,-19.238,-51.530,179.883,6.157,149.145
C09226=1102.413,-19.487,-51.516,179.883,6.153,149.144
C09227=1102.418,-19.737,-51.502,179.883,6.148,149.143
C09228=1102.423,-19.987,-51.488,179.882,6.143,149.142
C09229=1102.429,-20.236,-51.474,179.882,6.139,149.141
C09230=1102.433,-20.486,-51.460,179.882,6.133,149.140
C09231=1102.439,-20.735,-51.447,179.882,6.129,149.139
C09232=1102.444,-20.985,-51.433,179.881,6.125,149.138
C09233=1102.449,-21.235,-51.419,179.881,6.120,149.137
C09234=1102.454,-21.484,-51.406,179.880,6.115,149.136
C09235=1102.459,-21.734,-51.392,179.880,6.111,149.135
C09236=1102.464,-21.983,-51.378,179.880,6.107,149.134
C09237=1102.469,-22.233,-51.365,179.880,6.102,149.134
C09238=1102.474,-22.482,-51.351,179.880,6.097,149.132
C09239=1102.479,-22.731,-51.337,179.879,6.092,149.131
C09240=1102.484,-22.981,-51.324,179.879,6.088,149.131
C09241=1102.489,-23.231,-51.309,179.879,6.083,149.130
C09242=1102.495,-23.481,-51.296,179.878,6.079,149.129
C09243=1102.499,-23.730,-51.283,179.878,6.074,149.128
C09244=1102.505,-23.979,-51.269,179.878,6.070,149.127
C09245=1102.510,-24.229,-51.255,179.878,6.065,149.126
C09246=1102.514,-24.479,-51.241,179.877,6.060,149.125
C09247=1102.520,-24.728,-51.228,179.877,6.056,149.124
C09248=1102.525,-24.978,-51.214,179.877,6.050,149.123
C09249=1102.530,-25.227,-51.201,179.877,6.046,149.122
C09250=1102.535,-25.477,-51.187,179.877,6.042,149.121
C09251=1102.540,-25.728,-51.174,179.877,6.037,149.120
C09252=1102.545,-25.976,-51.160,179.876,6.032,149.119
C09253=1102.550,-26.227,-51.147,179.876,6.027,149.118
C09254=1102.555,-26.475,-51.133,179.875,6.022,149.117
C09255=1102.560,-26.726,-51.120,179.875,6.019,149.116
C09256=1102.566,-26.975,-51.106,179.875,6.014,149.115
C09257=1102.570,-27.225,-51.093,179.874,6.009,149.114
C09258=1102.576,-27.474,-51.079,179.874,6.004,149.114
C09259=1102.580,-27.724,-51.066,179.873,6.000,149.113
C09260=1102.586,-27.973,-51.052,179.873,5.995,149.112
C09261=1102.591,-28.223,-51.039,179.873,5.991,149.111
C09262=1102.595,-28.472,-51.025,179.873,5.986,149.110
C09263=1102.601,-28.722,-51.012,179.872,5.982,149.109
C09264=1102.606,-28.972,-50.999,179.872,5.977,149.108
C09265=1102.611,-29.221,-50.985,179.871,5.972,149.107
C09266=1102.616,-29.471,-50.972,179.871,5.968,149.106
C09267=1102.622,-29.720,-50.958,179.871,5.963,149.105
C09268=1102.626,-29.970,-50.945,179.870,5.959,149.104
C09269=1102.632,-30.220,-50.932,179.870,5.954,149.104
C09270=1102.636,-30.469,-50.918,179.870,5.950,149.103
C09271=1102.642,-30.719,-50.905,179.870,5.945,149.102
C09272=1102.646,-30.932,-50.893,179.869,5.942,149.101
C09273=1102.650,-31.147,-50.882,179.869,5.938,149.100
C09274=1102.654,-31.361,-50.871,179.869,5.933,149.099
C09275=1102.659,-31.575,-50.859,179.868,5.930,149.099
C09276=1102.663,-31.789,-50.847,179.868,5.926,149.098
